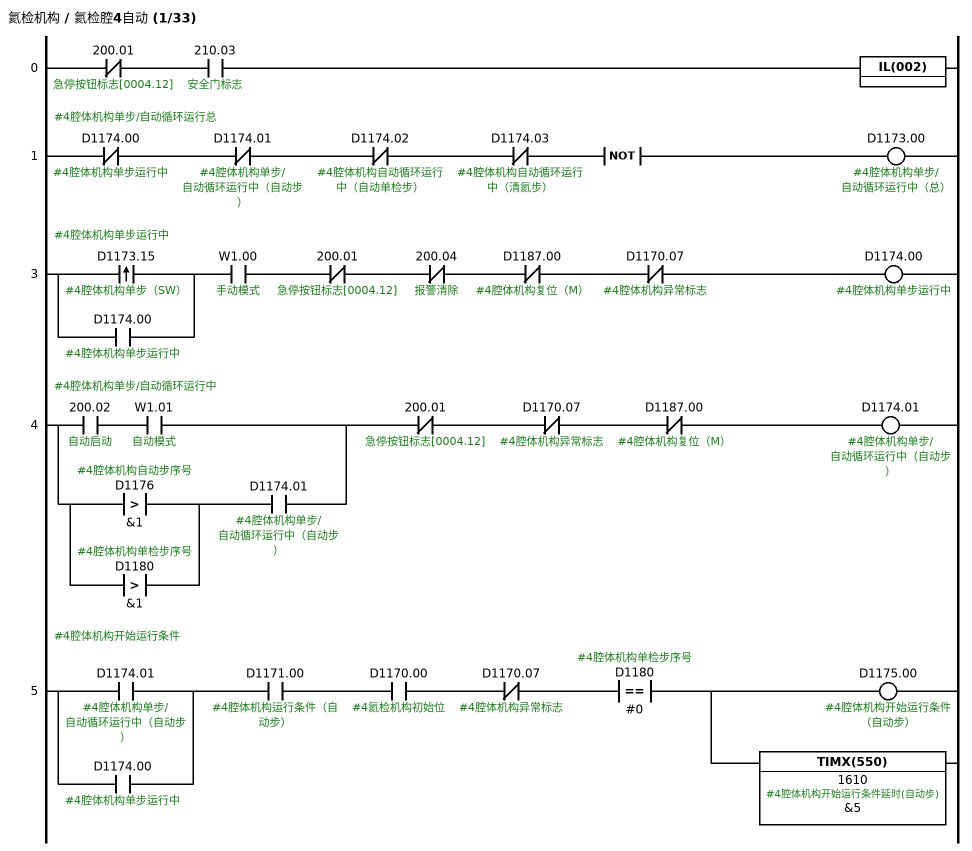
; [picture p336: 氦检机构 / 氦检腔4自动, rungs 0-5]
; rung 0
LDNOT 200.01  ; 急停按钮标志[0004.12]
AND 210.03  ; 安全门标志
IL(002)
; rung 1: #4腔体机构单步/自动循环运行总
LDNOT D1174.00  ; #4腔体机构单步运行中
ANDNOT D1174.01  ; #4腔体机构单步/自动循环运行中（自动步）
ANDNOT D1174.02  ; #4腔体机构自动循环运行中（自动单检步）
ANDNOT D1174.03  ; #4腔体机构自动循环运行中（清氦步）
NOT(520)
OUT D1173.00  ; #4腔体机构单步/自动循环运行中（总）
; rung 2: ******************************* / 自动双检步序 / *******************************
; rung 3: #4腔体机构单步运行中
@LD D1173.15  ; #4腔体机构单步（SW）
OR D1174.00  ; #4腔体机构单步运行中
AND W1.00  ; 手动模式
ANDNOT 200.01  ; 急停按钮标志[0004.12]
ANDNOT 200.04  ; 报警清除
ANDNOT D1187.00  ; #4腔体机构复位（M）
ANDNOT D1170.07  ; #4腔体机构异常标志
OUT D1174.00  ; #4腔体机构单步运行中
; rung 4: #4腔体机构单步/自动循环运行中
LD 200.02  ; 自动启动
AND W1.01  ; 自动模式
LD>L(321) D1176 &1  ; #4腔体机构自动步序号
OR>L(321) D1180 &1  ; #4腔体机构单检步序号
AND D1174.01  ; #4腔体机构单步/自动循环运行中（自动步）
ORLD
ANDNOT 200.01  ; 急停按钮标志[0004.12]
ANDNOT D1170.07  ; #4腔体机构异常标志
ANDNOT D1187.00  ; #4腔体机构复位（M）
OUT D1174.01  ; #4腔体机构单步/自动循环运行中（自动步）
; rung 5: #4腔体机构开始运行条件
LD D1174.01  ; #4腔体机构单步/自动循环运行中（自动步）
OR D1174.00  ; #4腔体机构单步运行中
AND D1171.00  ; #4腔体机构运行条件（自动步）
AND D1170.00  ; #4氦检机构初始位
ANDNOT D1170.07  ; #4腔体机构异常标志
AND=L(301) D1180 #0  ; #4腔体机构单检步序号
OUT D1175.00  ; #4腔体机构开始运行条件（自动步）
TIMX(550) 1610 &5  ; #4腔体机构开始运行条件延时(自动步)

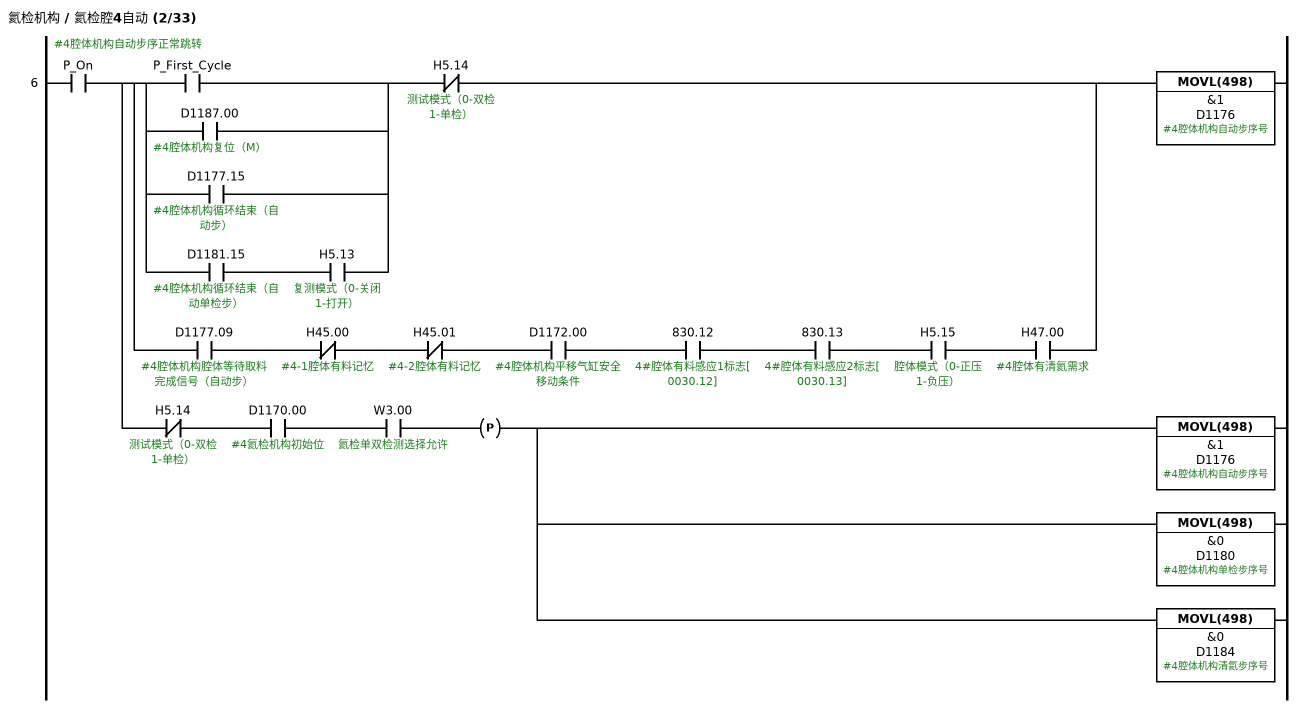
; rung 6: #4腔体机构自动步序正常跳转
LD P_On
OUT TR0
LD P_First_Cycle
OR D1187.00  ; #4腔体机构复位（M）
OR D1177.15  ; #4腔体机构循环结束（自动步）
LD D1181.15  ; #4腔体机构循环结束（自动单检步）
AND H5.13  ; 复测模式（0-关闭 1-打开）
ORLD
ANDNOT H5.14  ; 测试模式（0-双检 1-单检）
LD D1177.09  ; #4腔体机构腔体等待取料完成信号（自动步）  // 负压有清氦需求时，无需回初始位,直接跳回初始步序（D1176.00）
ANDNOT H45.00  ; #4-1腔体有料记忆
ANDNOT H45.01  ; #4-2腔体有料记忆
AND D1172.00  ; #4腔体机构平移气缸安全移动条件
AND 830.12  ; 4#腔体有料感应1标志[0030.12]
AND 830.13  ; 4#腔体有料感应2标志[0030.13]
AND H5.15  ; 腔体模式（0-正压 1-负压）
AND H47.00  ; #4腔体有清氦需求
ORLD
ANDLD
MOVL(498) &1 D1176  ; #4腔体机构自动步序号
LD TR0
ANDNOT H5.14  ; 测试模式（0-双检 1-单检）
AND D1170.00  ; #4氦检机构初始位
AND W3.00  ; 氦检单双检测选择允许
UP(521)
MOVL(498) &1 D1176  ; #4腔体机构自动步序号
MOVL(498) &0 D1180  ; #4腔体机构单检步序号
MOVL(498) &0 D1184  ; #4腔体机构清氦步序号

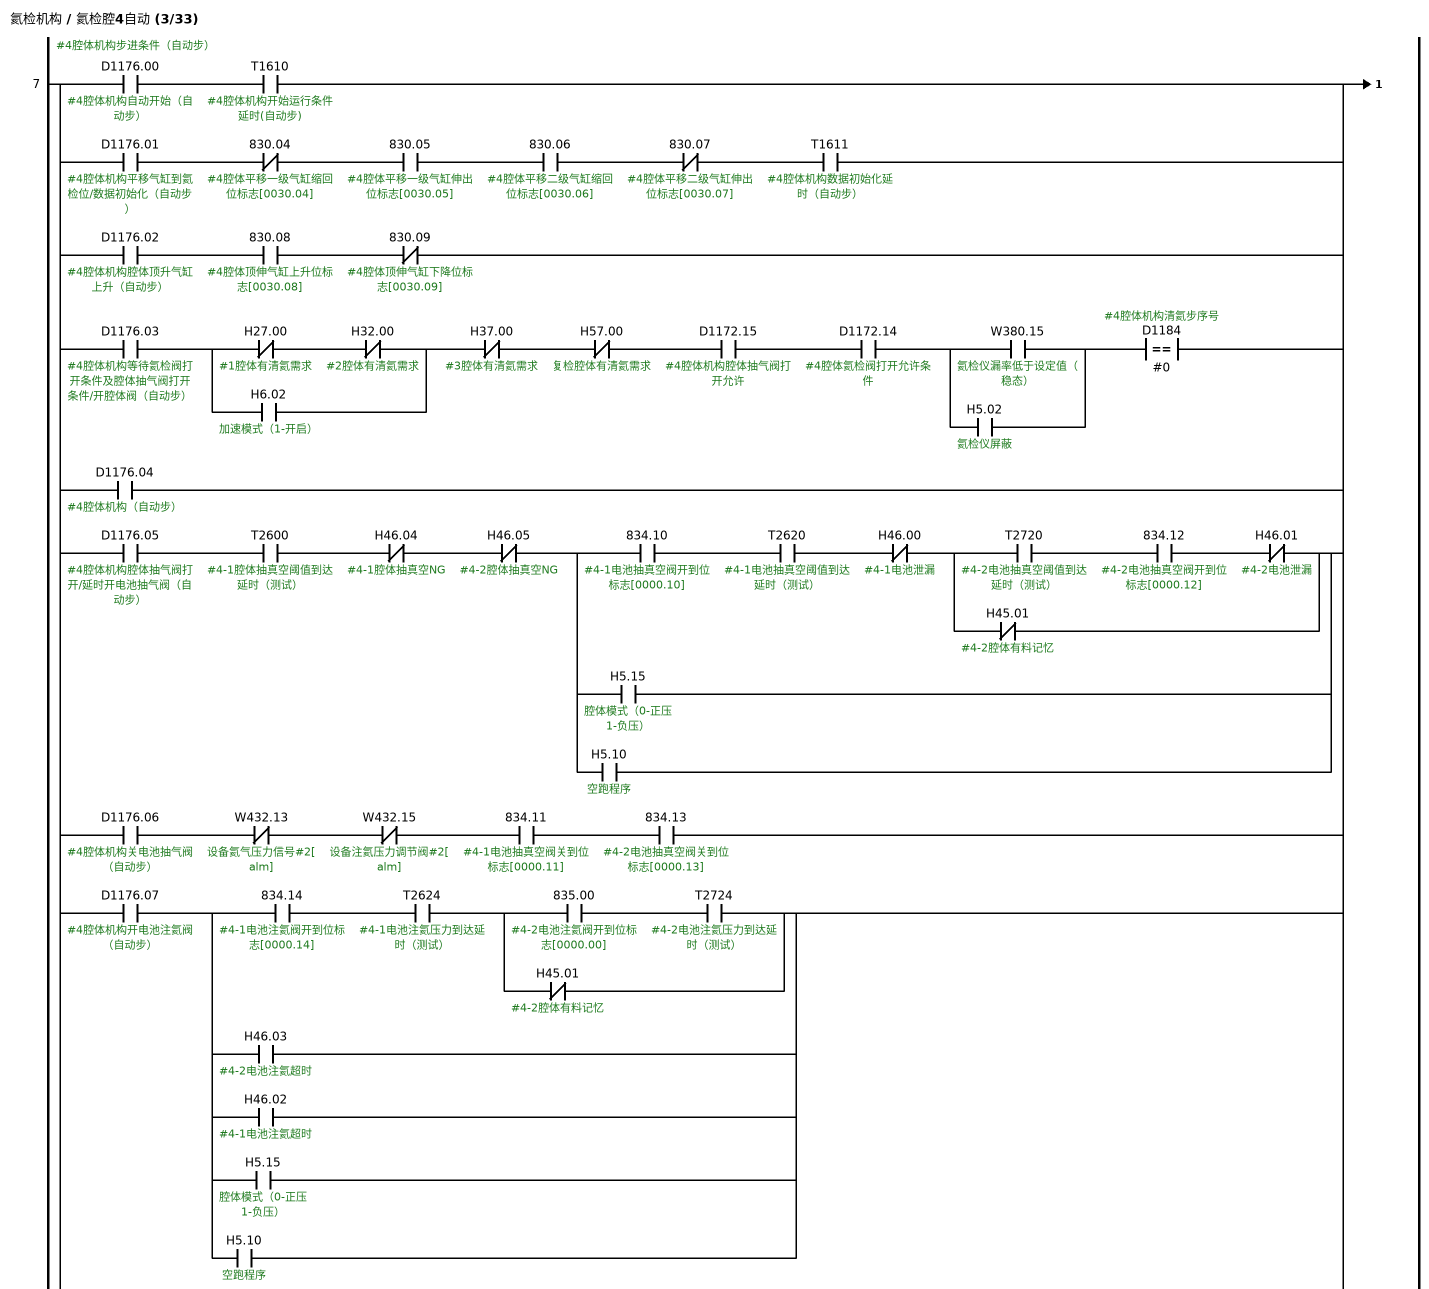

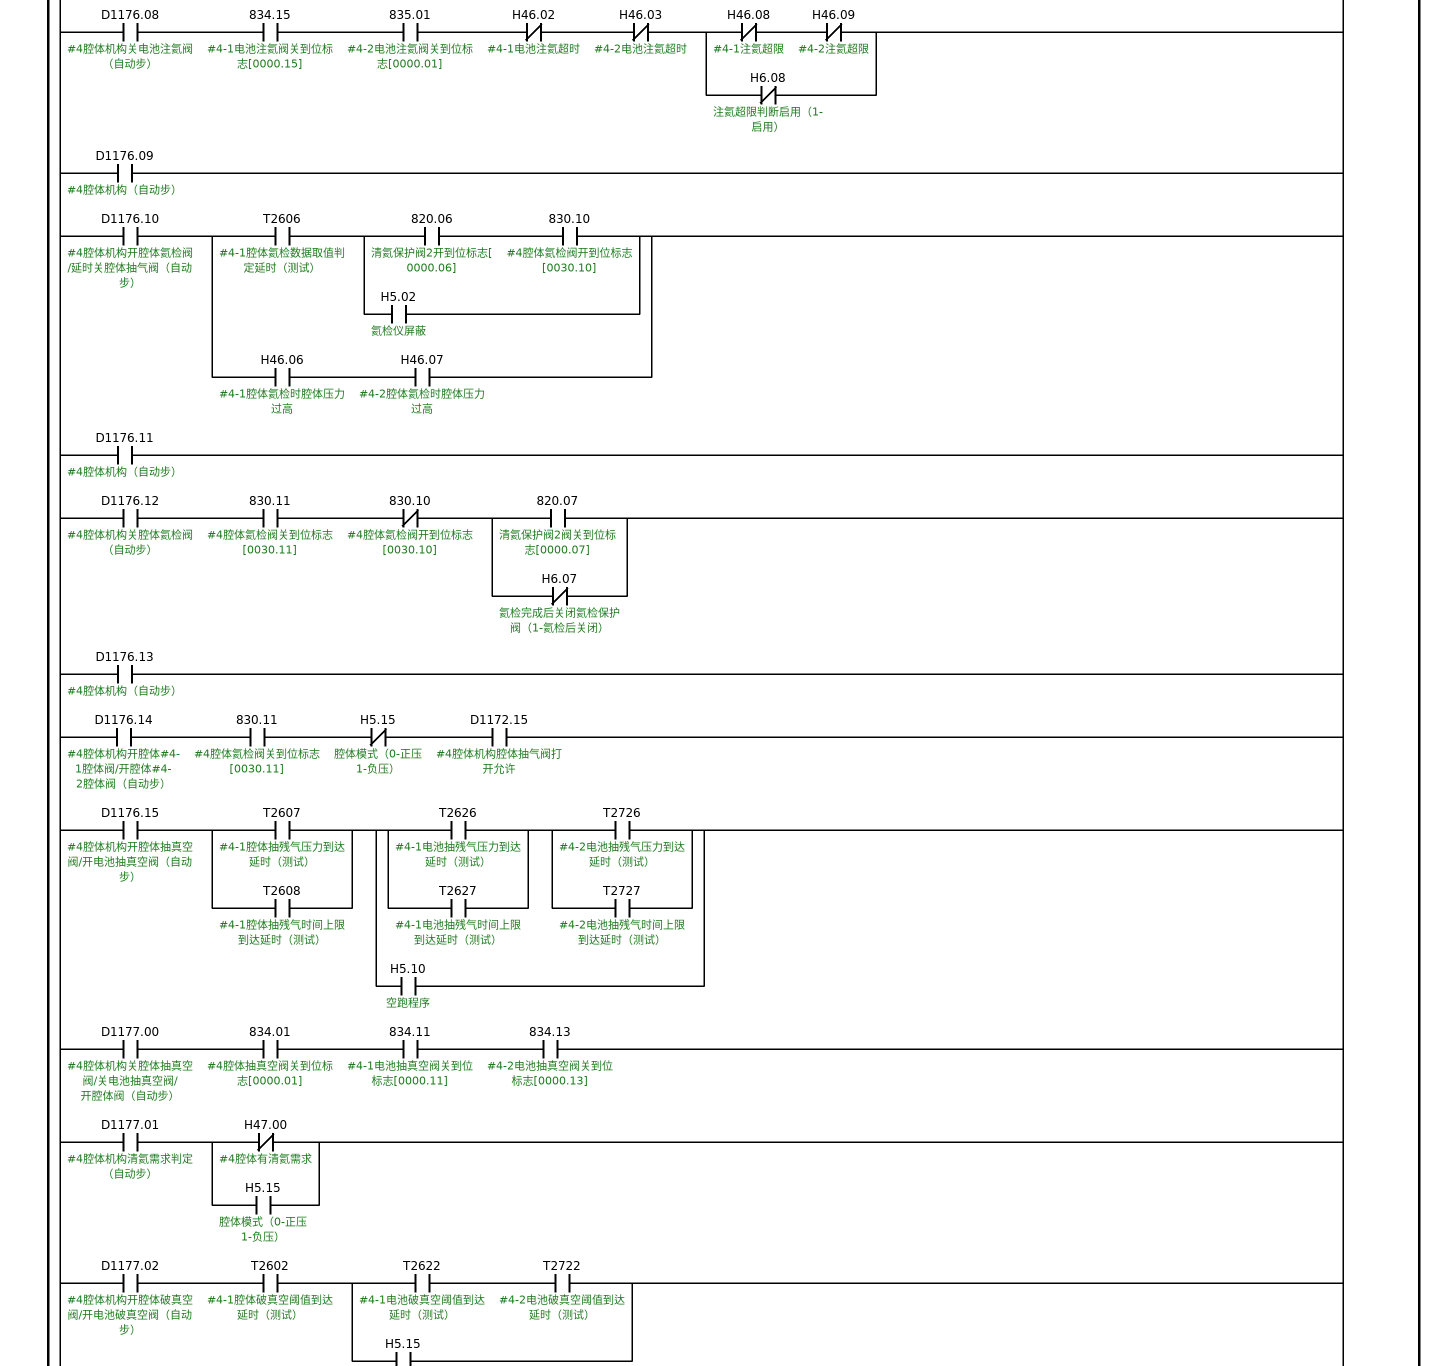

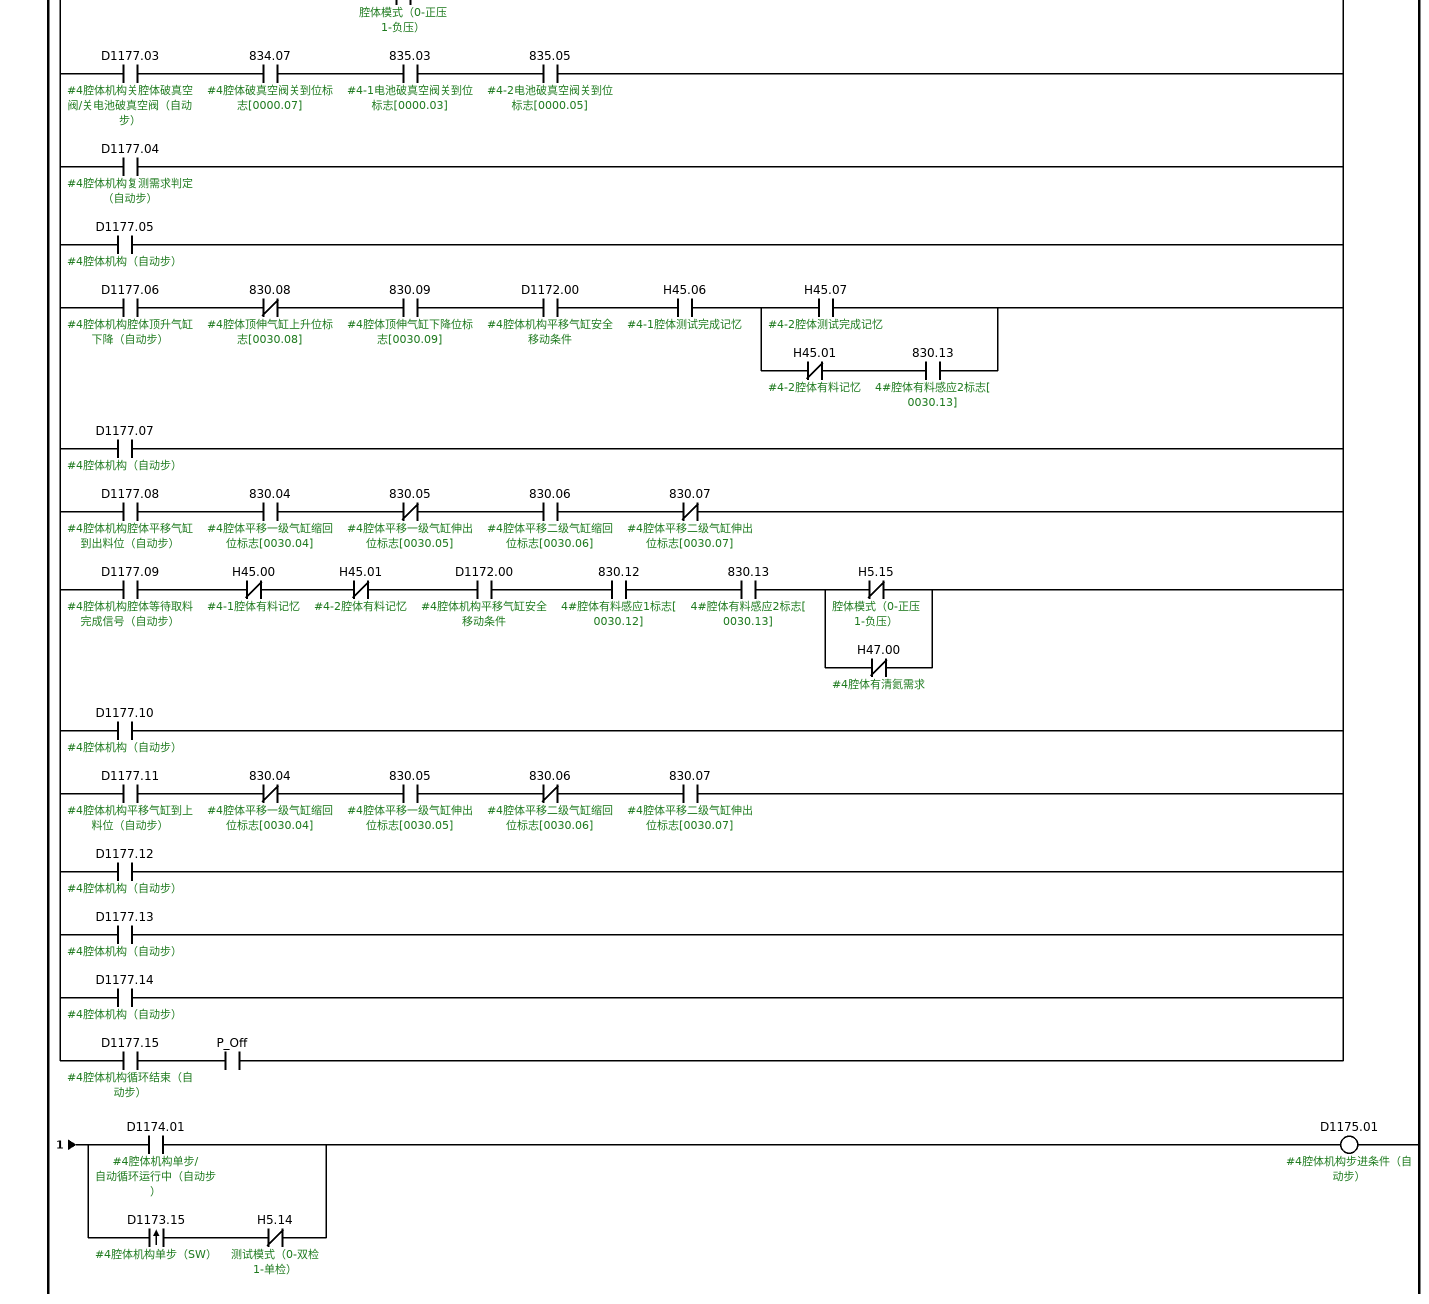
; rung 7: #4腔体机构步进条件（自动步）
LD D1176.00  ; #4腔体机构自动开始（自动步）
AND T1610  ; #4腔体机构开始运行条件延时(自动步)
LD D1176.01  ; #4腔体机构平移气缸到氦检位/数据初始化（自动步）
ANDNOT 830.04  ; #4腔体平移一级气缸缩回位标志[0030.04]
AND 830.05  ; #4腔体平移一级气缸伸出位标志[0030.05]
AND 830.06  ; #4腔体平移二级气缸缩回位标志[0030.06]
ANDNOT 830.07  ; #4腔体平移二级气缸伸出位标志[0030.07]
AND T1611  ; #4腔体机构数据初始化延时（自动步）
ORLD
LD D1176.02  ; #4腔体机构腔体顶升气缸上升（自动步）
AND 830.08  ; #4腔体顶伸气缸上升位标志[0030.08]
ANDNOT 830.09  ; #4腔体顶伸气缸下降位标志[0030.09]
ORLD
LD D1176.03  ; #4腔体机构等待氦检阀打开条件及腔体抽气阀打开条件/开腔体阀（自动步）
LDNOT H27.00  ; #1腔体有清氦需求
ANDNOT H32.00  ; #2腔体有清氦需求
OR H6.02  ; 加速模式（1-开启）
ANDLD
ANDNOT H37.00  ; #3腔体有清氦需求
ANDNOT H57.00  ; 复检腔体有清氦需求
AND D1172.15  ; #4腔体机构腔体抽气阀打开允许
AND D1172.14  ; #4腔体氦检阀打开允许条件
LD W380.15  ; 氦检仪漏率低于设定值（稳态）
OR H5.02  ; 氦检仪屏蔽
ANDLD
AND=L(301) D1184 #0  ; #4腔体机构清氦步序号
ORLD
OR D1176.04  ; #4腔体机构（自动步）
LD D1176.05  ; #4腔体机构腔体抽气阀打开/延时开电池抽气阀（自动步）
AND T2600  ; #4-1腔体抽真空阈值到达延时（测试）
ANDNOT H46.04  ; #4-1腔体抽真空NG
ANDNOT H46.05  ; #4-2腔体抽真空NG
LD 834.10  ; #4-1电池抽真空阀开到位标志[0000.10]
AND T2620  ; #4-1电池抽真空阈值到达延时（测试）
ANDNOT H46.00  ; #4-1电池泄漏
LD T2720  ; #4-2电池抽真空阈值到达延时（测试）
AND 834.12  ; #4-2电池抽真空阀开到位标志[0000.12]
ANDNOT H46.01  ; #4-2电池泄漏
ORNOT H45.01  ; #4-2腔体有料记忆
ANDLD
OR H5.15  ; 腔体模式（0-正压 1-负压）
OR H5.10  ; 空跑程序
ANDLD
ORLD
LD D1176.06  ; #4腔体机构关电池抽气阀（自动步）  // 单个电池出现电池泄漏时，需将对应的腔体阀门关闭
ANDNOT W432.13  ; 设备氦气压力信号#2[alm]
ANDNOT W432.15  ; 设备注氦压力调节阀#2[alm]
AND 834.11  ; #4-1电池抽真空阀关到位标志[0000.11]
AND 834.13  ; #4-2电池抽真空阀关到位标志[0000.13]
ORLD
LD D1176.07  ; #4腔体机构开电池注氦阀（自动步）  // 单个电池出现注氦超时时，需将对应的腔体阀门关闭
LD 834.14  ; #4-1电池注氦阀开到位标志[0000.14]
AND T2624  ; #4-1电池注氦压力到达延时（测试）
LD 835.00  ; #4-2电池注氦阀开到位标志[0000.00]
AND T2724  ; #4-2电池注氦压力到达延时（测试）
ORNOT H45.01  ; #4-2腔体有料记忆
ANDLD
OR H46.03  ; #4-2电池注氦超时
OR H46.02  ; #4-1电池注氦超时
OR H5.15  ; 腔体模式（0-正压 1-负压）
OR H5.10  ; 空跑程序
ANDLD
ORLD
LD D1176.08  ; #4腔体机构关电池注氦阀（自动步）
AND 834.15  ; #4-1电池注氦阀关到位标志[0000.15]
AND 835.01  ; #4-2电池注氦阀关到位标志[0000.01]
ANDNOT H46.02  ; #4-1电池注氦超时
ANDNOT H46.03  ; #4-2电池注氦超时
LDNOT H46.08  ; #4-1注氦超限
ANDNOT H46.09  ; #4-2注氦超限
ORNOT H6.08  ; 注氦超限判断启用（1-启用）
ANDLD
ORLD
OR D1176.09  ; #4腔体机构（自动步）
LD D1176.10  ; #4腔体机构开腔体氦检阀/延时关腔体抽气阀（自动步）
LD T2606  ; #4-1腔体氦检数据取值判定延时（测试）
LD 820.06  ; 清氦保护阀2开到位标志[0000.06]
AND 830.10  ; #4腔体氦检阀开到位标志[0030.10]
OR H5.02  ; 氦检仪屏蔽
ANDLD
LD H46.06  ; #4-1腔体氦检时腔体压力过高
AND H46.07  ; #4-2腔体氦检时腔体压力过高
ORLD
ANDLD
ORLD
OR D1176.11  ; #4腔体机构（自动步）
LD D1176.12  ; #4腔体机构关腔体氦检阀（自动步）
AND 830.11  ; #4腔体氦检阀关到位标志[0030.11]
ANDNOT 830.10  ; #4腔体氦检阀开到位标志[0030.10]
LD 820.07  ; 清氦保护阀2阀关到位标志[0000.07]
ORNOT H6.07  ; 氦检完成后关闭氦检保护阀（1-氦检后关闭）
ANDLD
ORLD
OR D1176.13  ; #4腔体机构（自动步）
LD D1176.14  ; #4腔体机构开腔体#4-1腔体阀/开腔体#4-2腔体阀（自动步）
AND 830.11  ; #4腔体氦检阀关到位标志[0030.11]
ANDNOT H5.15  ; 腔体模式（0-正压 1-负压）
AND D1172.15  ; #4腔体机构腔体抽气阀打开允许
ORLD
LD D1176.15  ; #4腔体机构开腔体抽真空阀/开电池抽真空阀（自动步）
LD T2607  ; #4-1腔体抽残气压力到达延时（测试）
OR T2608  ; #4-1腔体抽残气时间上限到达延时（测试）
ANDLD
LD T2626  ; #4-1电池抽残气压力到达延时（测试）
OR T2627  ; #4-1电池抽残气时间上限到达延时（测试）
LD T2726  ; #4-2电池抽残气压力到达延时（测试）
OR T2727  ; #4-2电池抽残气时间上限到达延时（测试）
ANDLD
OR H5.10  ; 空跑程序
ANDLD
ORLD
LD D1177.00  ; #4腔体机构关腔体抽真空阀/关电池抽真空阀/开腔体阀（自动步）
AND 834.01  ; #4腔体抽真空阀关到位标志[0000.01]
AND 834.11  ; #4-1电池抽真空阀关到位标志[0000.11]
AND 834.13  ; #4-2电池抽真空阀关到位标志[0000.13]
ORLD
LD D1177.01  ; #4腔体机构清氦需求判定（自动步）
LDNOT H47.00  ; #4腔体有清氦需求
OR H5.15  ; 腔体模式（0-正压 1-负压）
ANDLD
ORLD
LD D1177.02  ; #4腔体机构开腔体破真空阀/开电池破真空阀（自动步）
AND T2602  ; #4-1腔体破真空阈值到达延时（测试）
LD T2622  ; #4-1电池破真空阈值到达延时（测试）
AND T2722  ; #4-2电池破真空阈值到达延时（测试）
OR H5.15  ; 腔体模式（0-正压 1-负压）
ANDLD
ORLD
LD D1177.03  ; #4腔体机构关腔体破真空阀/关电池破真空阀（自动步）
AND 834.07  ; #4腔体破真空阀关到位标志[0000.07]
AND 835.03  ; #4-1电池破真空阀关到位标志[0000.03]
AND 835.05  ; #4-2电池破真空阀关到位标志[0000.05]
ORLD
OR D1177.04  ; #4腔体机构复测需求判定（自动步）
OR D1177.05  ; #4腔体机构（自动步）
LD D1177.06  ; #4腔体机构腔体顶升气缸下降（自动步）
ANDNOT 830.08  ; #4腔体顶伸气缸上升位标志[0030.08]
AND 830.09  ; #4腔体顶伸气缸下降位标志[0030.09]
AND D1172.00  ; #4腔体机构平移气缸安全移动条件
AND H45.06  ; #4-1腔体测试完成记忆
LD H45.07  ; #4-2腔体测试完成记忆
LDNOT H45.01  ; #4-2腔体有料记忆
AND 830.13  ; 4#腔体有料感应2标志[0030.13]
ORLD
ANDLD
ORLD
OR D1177.07  ; #4腔体机构（自动步）
LD D1177.08  ; #4腔体机构腔体平移气缸到出料位（自动步）
AND 830.04  ; #4腔体平移一级气缸缩回位标志[0030.04]
ANDNOT 830.05  ; #4腔体平移一级气缸伸出位标志[0030.05]
AND 830.06  ; #4腔体平移二级气缸缩回位标志[0030.06]
ANDNOT 830.07  ; #4腔体平移二级气缸伸出位标志[0030.07]
ORLD
LD D1177.09  ; #4腔体机构腔体等待取料完成信号（自动步）  // 负压有清氦需求时，无需回初始位,直接跳回初始步序（D1176.00）
ANDNOT H45.00  ; #4-1腔体有料记忆
ANDNOT H45.01  ; #4-2腔体有料记忆
AND D1172.00  ; #4腔体机构平移气缸安全移动条件
AND 830.12  ; 4#腔体有料感应1标志[0030.12]
AND 830.13  ; 4#腔体有料感应2标志[0030.13]
LDNOT H5.15  ; 腔体模式（0-正压 1-负压）
ORNOT H47.00  ; #4腔体有清氦需求
ANDLD
ORLD
OR D1177.10  ; #4腔体机构（自动步）
LD D1177.11  ; #4腔体机构平移气缸到上料位（自动步）
ANDNOT 830.04  ; #4腔体平移一级气缸缩回位标志[0030.04]
AND 830.05  ; #4腔体平移一级气缸伸出位标志[0030.05]
ANDNOT 830.06  ; #4腔体平移二级气缸缩回位标志[0030.06]
AND 830.07  ; #4腔体平移二级气缸伸出位标志[0030.07]
ORLD
OR D1177.12  ; #4腔体机构（自动步）
OR D1177.13  ; #4腔体机构（自动步）
OR D1177.14  ; #4腔体机构（自动步）
LD D1177.15  ; #4腔体机构循环结束（自动步）
AND P_Off
ORLD
LD D1174.01  ; #4腔体机构单步/自动循环运行中（自动步）
@LD D1173.15  ; #4腔体机构单步（SW）
ANDNOT H5.14  ; 测试模式（0-双检 1-单检）
ORLD
ANDLD
OUT D1175.01  ; #4腔体机构步进条件（自动步）

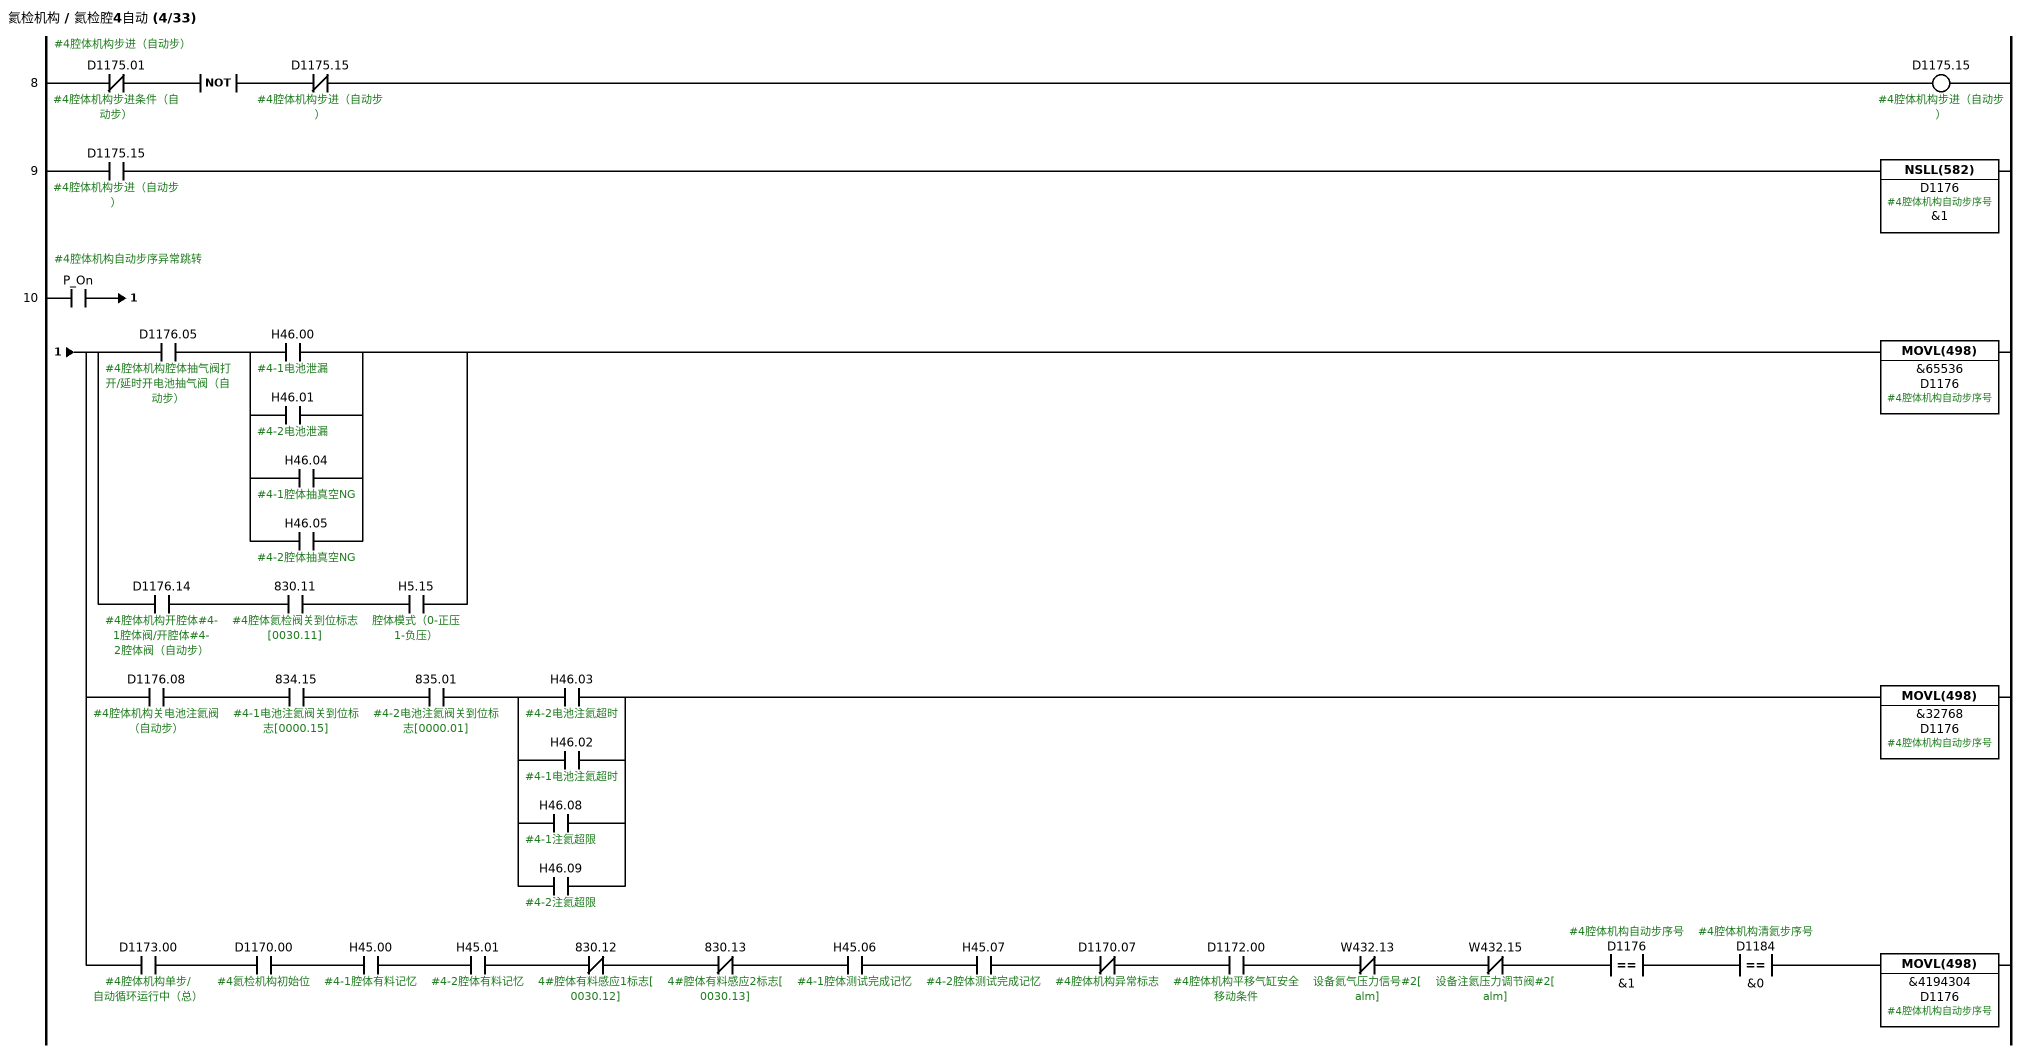
; rung 8: #4腔体机构步进（自动步）
LDNOT D1175.01  ; #4腔体机构步进条件（自动步）
NOT(520)
ANDNOT D1175.15  ; #4腔体机构步进（自动步）
OUT D1175.15  ; #4腔体机构步进（自动步）
; rung 9
LD D1175.15  ; #4腔体机构步进（自动步）
NSLL(582) D1176 &1  ; #4腔体机构自动步序号
; rung 10: #4腔体机构自动步序异常跳转
LD P_On
OUT TR0
LD D1176.05  ; #4腔体机构腔体抽气阀打开/延时开电池抽气阀（自动步）
LD H46.00  ; #4-1电池泄漏
OR H46.01  ; #4-2电池泄漏
OR H46.04  ; #4-1腔体抽真空NG
OR H46.05  ; #4-2腔体抽真空NG
ANDLD
LD D1176.14  ; #4腔体机构开腔体#4-1腔体阀/开腔体#4-2腔体阀（自动步）  // 负压模式不需要进行氦检后抽真空动作
AND 830.11  ; #4腔体氦检阀关到位标志[0030.11]
AND H5.15  ; 腔体模式（0-正压 1-负压）
ORLD
ANDLD
MOVL(498) &65536 D1176  ; #4腔体机构自动步序号  // 出现腔体抽真空NG，双电池抽真空NG，均跳转至自动步序D1067.0
LD TR0
AND D1176.08  ; #4腔体机构关电池注氦阀（自动步）
AND 834.15  ; #4-1电池注氦阀关到位标志[0000.15]
AND 835.01  ; #4-2电池注氦阀关到位标志[0000.01]
LD H46.03  ; #4-2电池注氦超时
OR H46.02  ; #4-1电池注氦超时
OR H46.08  ; #4-1注氦超限
OR H46.09  ; #4-2注氦超限
ANDLD
MOVL(498) &32768 D1176  ; #4腔体机构自动步序号  // 注氦超时需跳转至清氦步序（D1176.15）
LD TR0
AND D1173.00  ; #4腔体机构单步/自动循环运行中（总）
AND D1170.00  ; #4氦检机构初始位
AND H45.00  ; #4-1腔体有料记忆
AND H45.01  ; #4-2腔体有料记忆
ANDNOT 830.12  ; 4#腔体有料感应1标志[0030.12]
ANDNOT 830.13  ; 4#腔体有料感应2标志[0030.13]
AND H45.06  ; #4-1腔体测试完成记忆
AND H45.07  ; #4-2腔体测试完成记忆
ANDNOT D1170.07  ; #4腔体机构异常标志
AND D1172.00  ; #4腔体机构平移气缸安全移动条件
ANDNOT W432.13  ; 设备氦气压力信号#2[alm]
ANDNOT W432.15  ; 设备注氦压力调节阀#2[alm]
AND=L(301) D1176 &1  ; #4腔体机构自动步序号
AND=L(301) D1184 &0  ; #4腔体机构清氦步序号
MOVL(498) &4194304 D1176  ; #4腔体机构自动步序号  // 带料复位时，腔体测试完成后直接跳转至D1177.06
; rung 11: ******************************* / 清氦步序 / *******************************

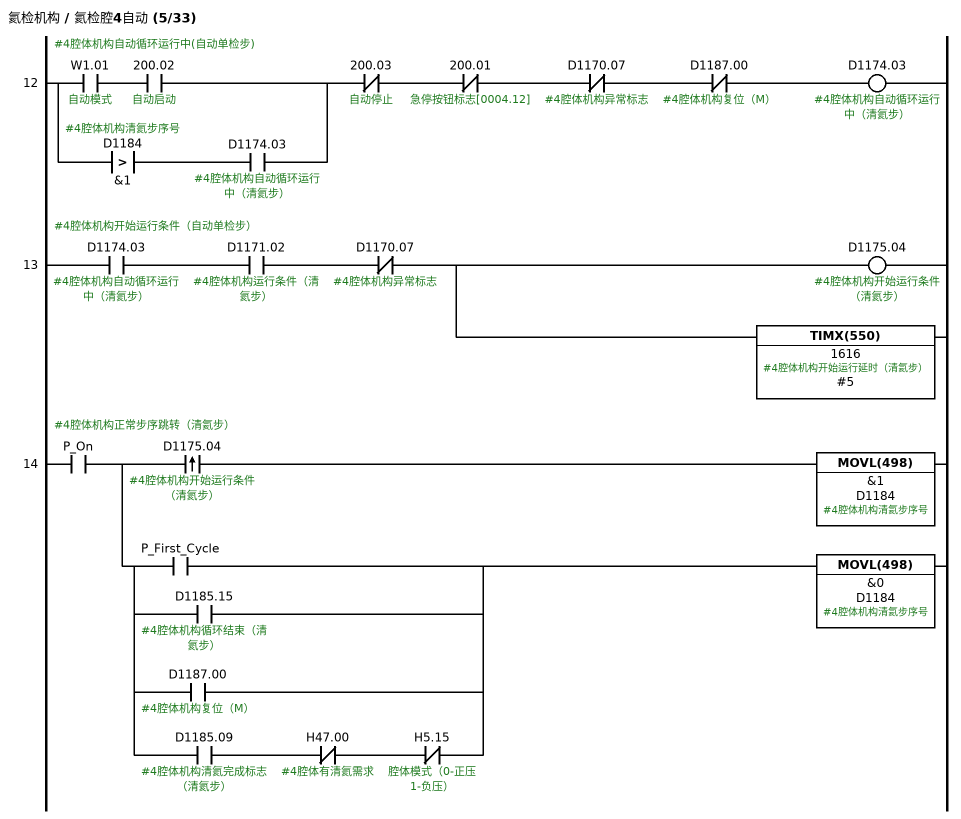
; rung 12: #4腔体机构自动循环运行中(自动单检步)
LD W1.01  ; 自动模式
AND 200.02  ; 自动启动
LD>L(321) D1184 &1  ; #4腔体机构清氦步序号
AND D1174.03  ; #4腔体机构自动循环运行中（清氦步）
ORLD
ANDNOT 200.03  ; 自动停止
ANDNOT 200.01  ; 急停按钮标志[0004.12]
ANDNOT D1170.07  ; #4腔体机构异常标志
ANDNOT D1187.00  ; #4腔体机构复位（M）
OUT D1174.03  ; #4腔体机构自动循环运行中（清氦步）
; rung 13: #4腔体机构开始运行条件（自动单检步）
LD D1174.03  ; #4腔体机构自动循环运行中（清氦步）
AND D1171.02  ; #4腔体机构运行条件（清氦步）
ANDNOT D1170.07  ; #4腔体机构异常标志
OUT D1175.04  ; #4腔体机构开始运行条件（清氦步）
TIMX(550) 1616 #5  ; #4腔体机构开始运行延时（清氦步）
; rung 14: #4腔体机构正常步序跳转（清氦步）
LD P_On
OUT TR0
@AND D1175.04  ; #4腔体机构开始运行条件（清氦步）
MOVL(498) &1 D1184  ; #4腔体机构清氦步序号
LD TR0
LD P_First_Cycle
OR D1185.15  ; #4腔体机构循环结束（清氦步）
OR D1187.00  ; #4腔体机构复位（M）
LD D1185.09  ; #4腔体机构清氦完成标志（清氦步）  // 正压腔体是待料清氦，需跳转回测试步序
ANDNOT H47.00  ; #4腔体有清氦需求
ANDNOT H5.15  ; 腔体模式（0-正压 1-负压）
ORLD
ANDLD
MOVL(498) &0 D1184  ; #4腔体机构清氦步序号

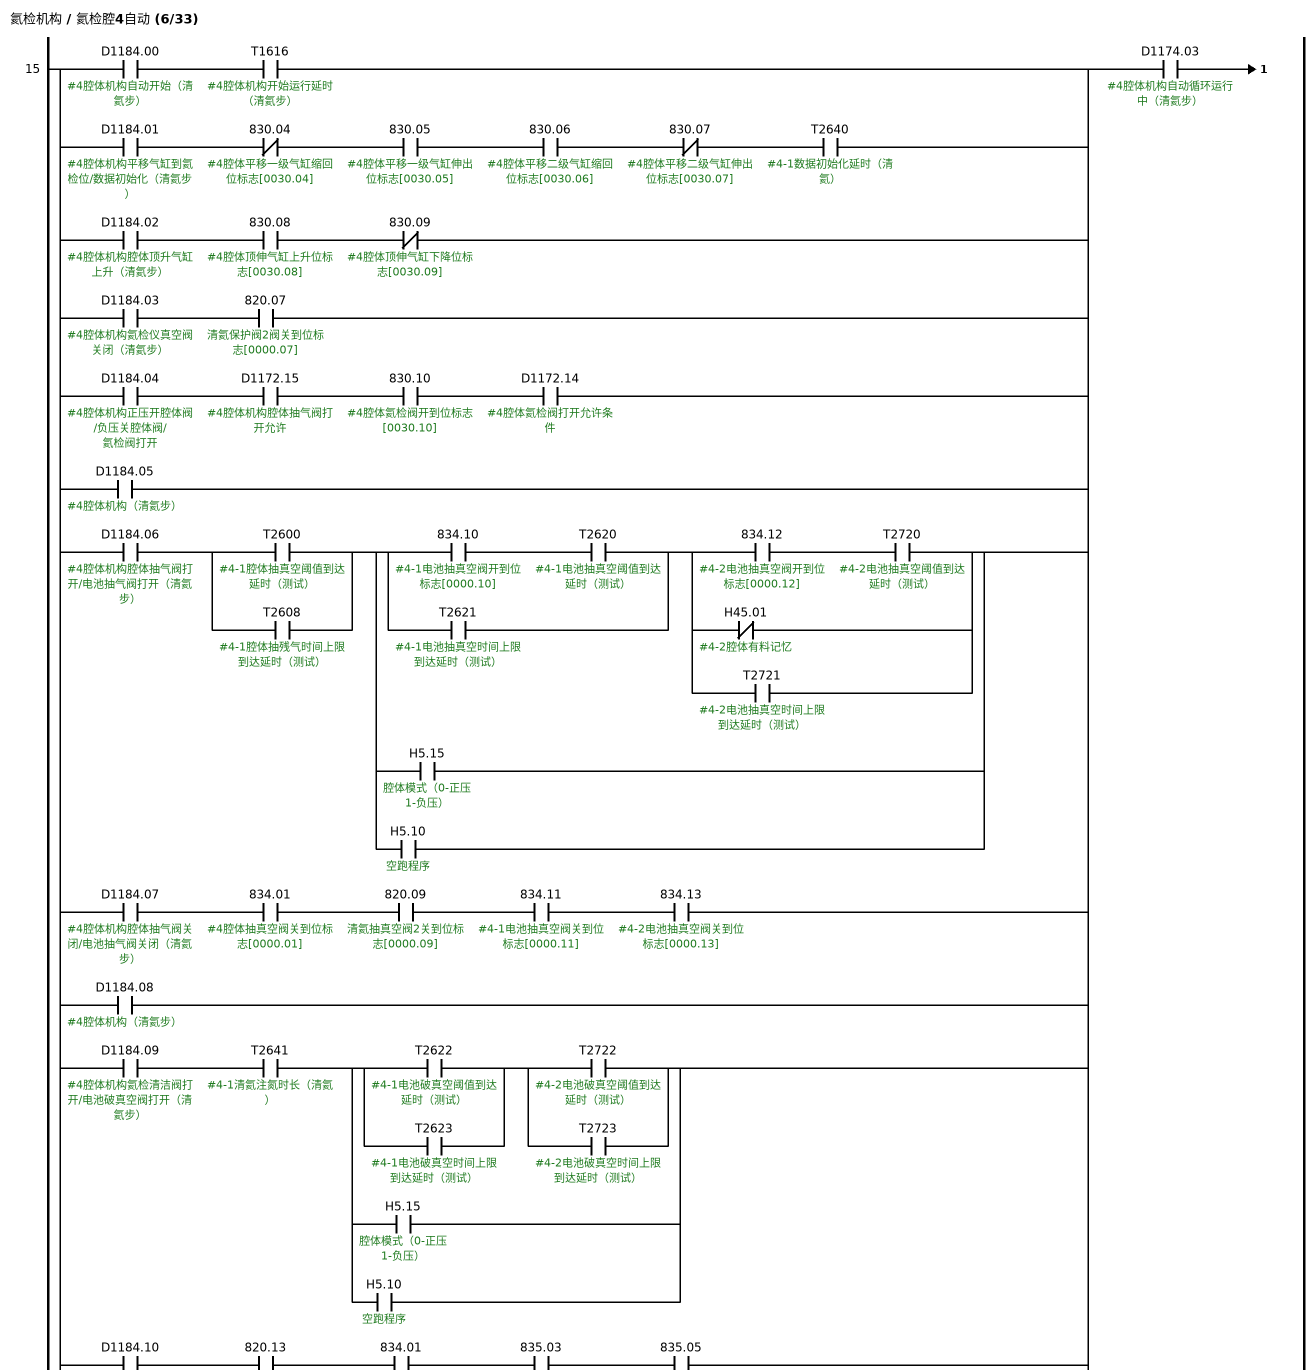

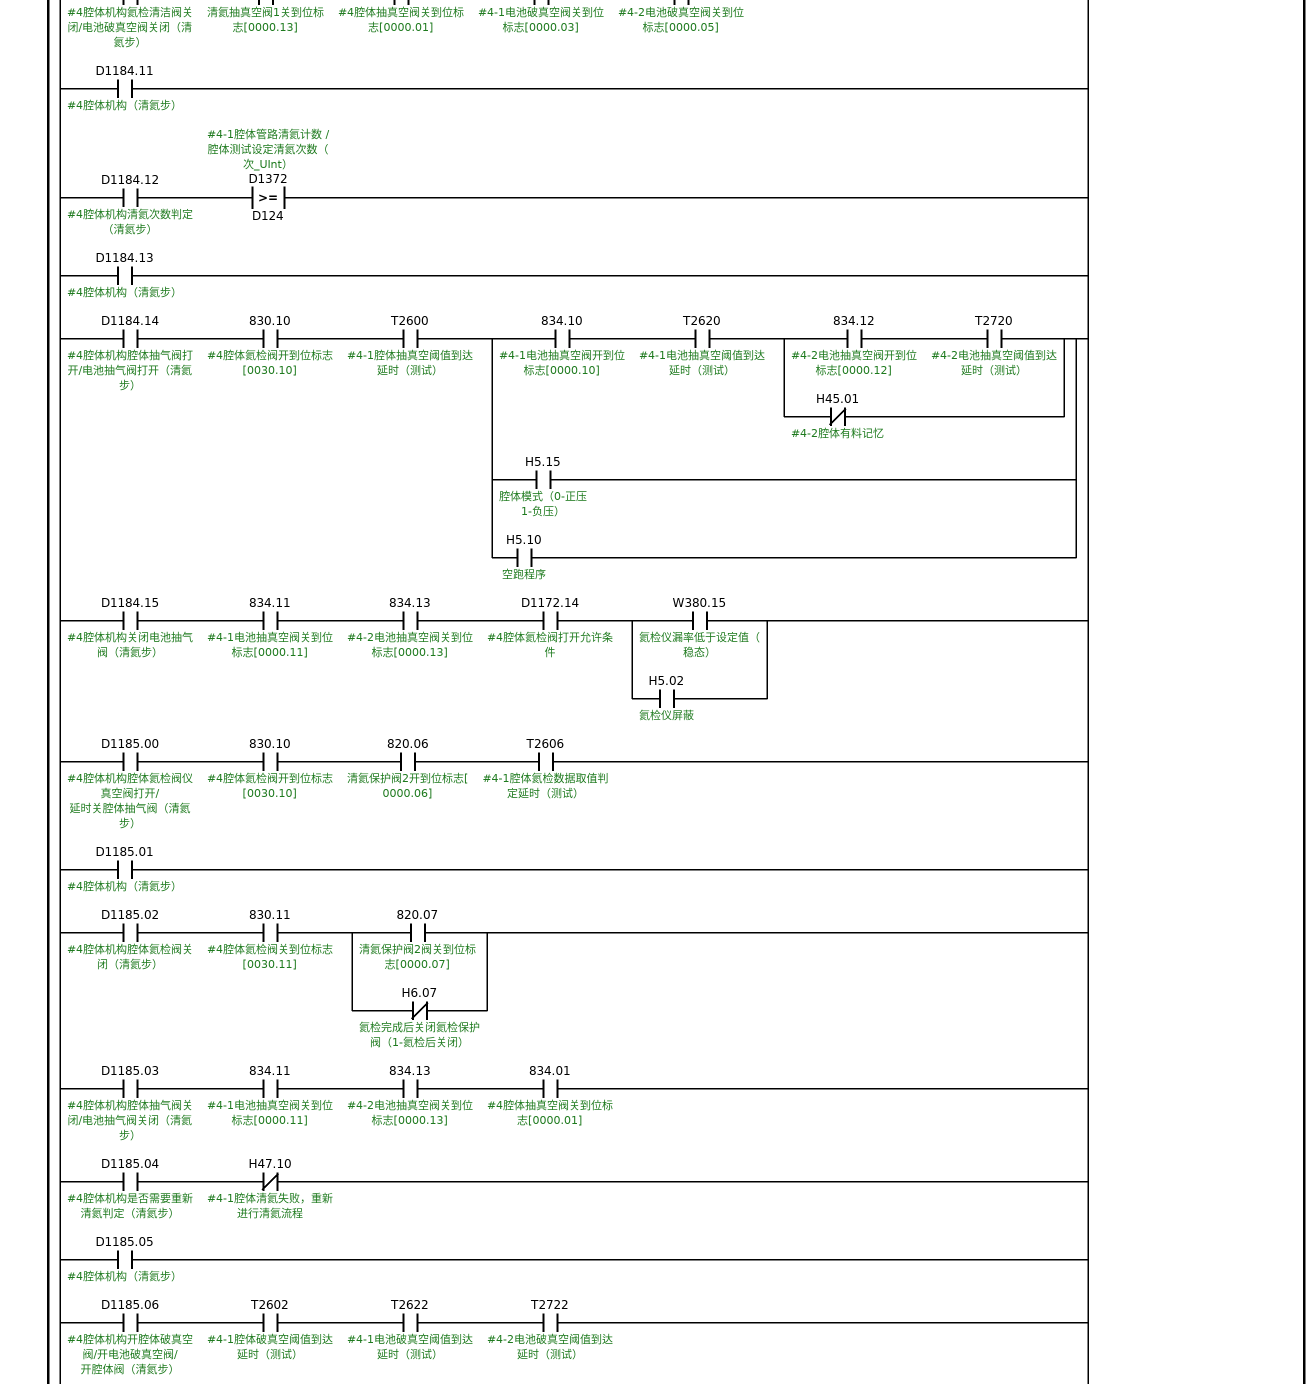

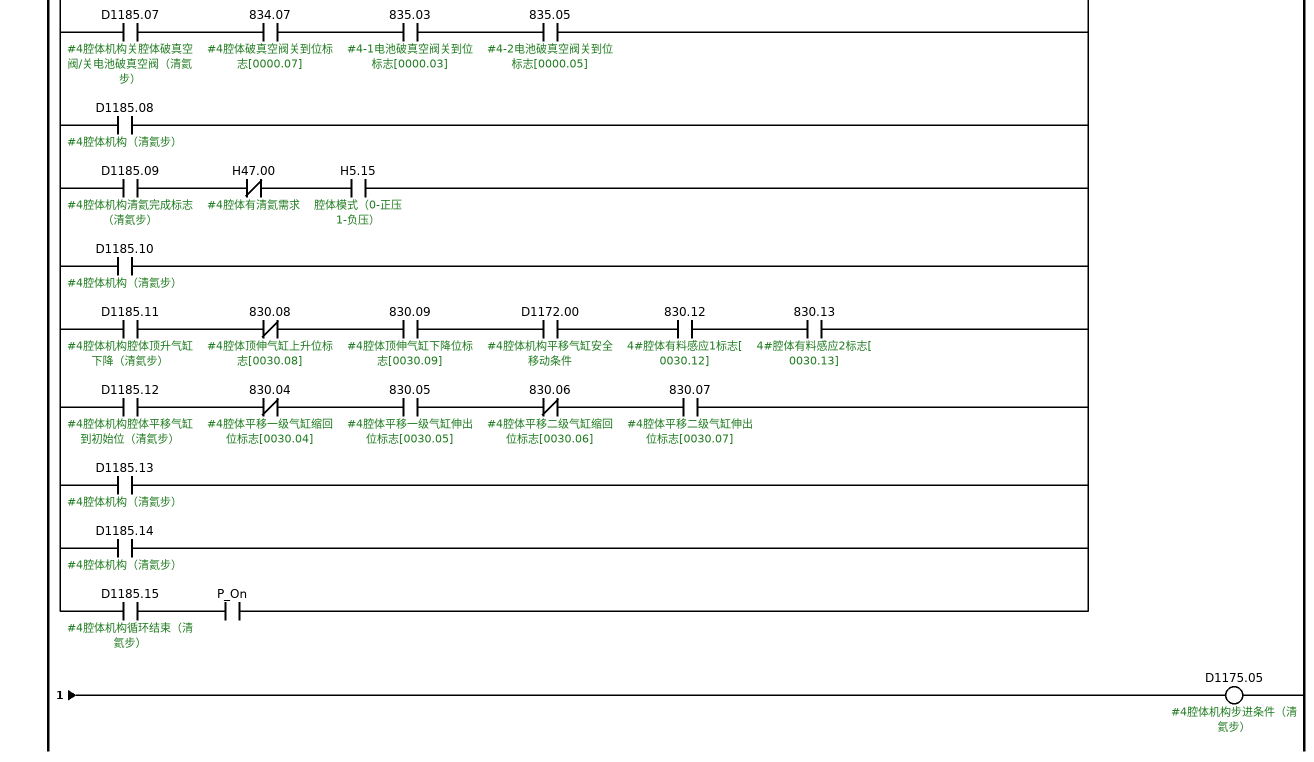
; rung 15
LD D1184.00  ; #4腔体机构自动开始（清氦步）
AND T1616  ; #4腔体机构开始运行延时（清氦步）
LD D1184.01  ; #4腔体机构平移气缸到氦检位/数据初始化（清氦步）
ANDNOT 830.04  ; #4腔体平移一级气缸缩回位标志[0030.04]
AND 830.05  ; #4腔体平移一级气缸伸出位标志[0030.05]
AND 830.06  ; #4腔体平移二级气缸缩回位标志[0030.06]
ANDNOT 830.07  ; #4腔体平移二级气缸伸出位标志[0030.07]
AND T2640  ; #4-1数据初始化延时（清氦）
ORLD
LD D1184.02  ; #4腔体机构腔体顶升气缸上升（清氦步）
AND 830.08  ; #4腔体顶伸气缸上升位标志[0030.08]
ANDNOT 830.09  ; #4腔体顶伸气缸下降位标志[0030.09]
ORLD
LD D1184.03  ; #4腔体机构氦检仪真空阀关闭（清氦步）
AND 820.07  ; 清氦保护阀2阀关到位标志[0000.07]
ORLD
LD D1184.04  ; #4腔体机构正压开腔体阀/负压关腔体阀/氦检阀打开  // 负压模式下，复测前的清氦不允许抽电池
AND D1172.15  ; #4腔体机构腔体抽气阀打开允许
AND 830.10  ; #4腔体氦检阀开到位标志[0030.10]
AND D1172.14  ; #4腔体氦检阀打开允许条件
ORLD
OR D1184.05  ; #4腔体机构（清氦步）
LD D1184.06  ; #4腔体机构腔体抽气阀打开/电池抽气阀打开（清氦步）
LD T2600  ; #4-1腔体抽真空阈值到达延时（测试）
OR T2608  ; #4-1腔体抽残气时间上限到达延时（测试）
ANDLD
LD 834.10  ; #4-1电池抽真空阀开到位标志[0000.10]
AND T2620  ; #4-1电池抽真空阈值到达延时（测试）
OR T2621  ; #4-1电池抽真空时间上限到达延时（测试）
LD 834.12  ; #4-2电池抽真空阀开到位标志[0000.12]
AND T2720  ; #4-2电池抽真空阈值到达延时（测试）
ORNOT H45.01  ; #4-2腔体有料记忆
OR T2721  ; #4-2电池抽真空时间上限到达延时（测试）
ANDLD
OR H5.15  ; 腔体模式（0-正压 1-负压）
OR H5.10  ; 空跑程序
ANDLD
ORLD
LD D1184.07  ; #4腔体机构腔体抽气阀关闭/电池抽气阀关闭（清氦步）
AND 834.01  ; #4腔体抽真空阀关到位标志[0000.01]
AND 820.09  ; 清氦抽真空阀2关到位标志[0000.09]
AND 834.11  ; #4-1电池抽真空阀关到位标志[0000.11]
AND 834.13  ; #4-2电池抽真空阀关到位标志[0000.13]
ORLD
OR D1184.08  ; #4腔体机构（清氦步）
LD D1184.09  ; #4腔体机构氦检清洁阀打开/电池破真空阀打开（清氦步）
AND T2641  ; #4-1清氦注氮时长（清氦）
LD T2622  ; #4-1电池破真空阈值到达延时（测试）
OR T2623  ; #4-1电池破真空时间上限到达延时（测试）
LD T2722  ; #4-2电池破真空阈值到达延时（测试）
OR T2723  ; #4-2电池破真空时间上限到达延时（测试）
ANDLD
OR H5.15  ; 腔体模式（0-正压 1-负压）
OR H5.10  ; 空跑程序
ANDLD
ORLD
LD D1184.10  ; #4腔体机构氦检清洁阀关闭/电池破真空阀关闭（清氦步）
AND 820.13  ; 清氦抽真空阀1关到位标志[0000.13]
AND 834.01  ; #4腔体抽真空阀关到位标志[0000.01]
AND 835.03  ; #4-1电池破真空阀关到位标志[0000.03]
AND 835.05  ; #4-2电池破真空阀关到位标志[0000.05]
ORLD
OR D1184.11  ; #4腔体机构（清氦步）
LD D1184.12  ; #4腔体机构清氦次数判定（清氦步）
AND>=(325) D1372 D124  ; #4-1腔体管路清氦计数, 腔体测试设定清氦次数（次_UInt）
ORLD
OR D1184.13  ; #4腔体机构（清氦步）
LD D1184.14  ; #4腔体机构腔体抽气阀打开/电池抽气阀打开（清氦步）
AND 830.10  ; #4腔体氦检阀开到位标志[0030.10]
AND T2600  ; #4-1腔体抽真空阈值到达延时（测试）
LD 834.10  ; #4-1电池抽真空阀开到位标志[0000.10]
AND T2620  ; #4-1电池抽真空阈值到达延时（测试）
LD 834.12  ; #4-2电池抽真空阀开到位标志[0000.12]
AND T2720  ; #4-2电池抽真空阈值到达延时（测试）
ORNOT H45.01  ; #4-2腔体有料记忆
ANDLD
OR H5.15  ; 腔体模式（0-正压 1-负压）
OR H5.10  ; 空跑程序
ANDLD
ORLD
LD D1184.15  ; #4腔体机构关闭电池抽气阀（清氦步）
AND 834.11  ; #4-1电池抽真空阀关到位标志[0000.11]
AND 834.13  ; #4-2电池抽真空阀关到位标志[0000.13]
AND D1172.14  ; #4腔体氦检阀打开允许条件
LD W380.15  ; 氦检仪漏率低于设定值（稳态）
OR H5.02  ; 氦检仪屏蔽
ANDLD
ORLD
LD D1185.00  ; #4腔体机构腔体氦检阀仪真空阀打开/延时关腔体抽气阀（清氦步）
AND 830.10  ; #4腔体氦检阀开到位标志[0030.10]
AND 820.06  ; 清氦保护阀2开到位标志[0000.06]
AND T2606  ; #4-1腔体氦检数据取值判定延时（测试）
ORLD
OR D1185.01  ; #4腔体机构（清氦步）
LD D1185.02  ; #4腔体机构腔体氦检阀关闭（清氦步）
AND 830.11  ; #4腔体氦检阀关到位标志[0030.11]
LD 820.07  ; 清氦保护阀2阀关到位标志[0000.07]
ORNOT H6.07  ; 氦检完成后关闭氦检保护阀（1-氦检后关闭）
ANDLD
ORLD
LD D1185.03  ; #4腔体机构腔体抽气阀关闭/电池抽气阀关闭（清氦步）
AND 834.11  ; #4-1电池抽真空阀关到位标志[0000.11]
AND 834.13  ; #4-2电池抽真空阀关到位标志[0000.13]
AND 834.01  ; #4腔体抽真空阀关到位标志[0000.01]
ORLD
LD D1185.04  ; #4腔体机构是否需要重新清氦判定（清氦步）
ANDNOT H47.10  ; #4-1腔体清氦失败，重新进行清氦流程  // 清氦失败，重新进行清氦
ORLD
OR D1185.05  ; #4腔体机构（清氦步）
LD D1185.06  ; #4腔体机构开腔体破真空阀/开电池破真空阀/开腔体阀（清氦步）
AND T2602  ; #4-1腔体破真空阈值到达延时（测试）
AND T2622  ; #4-1电池破真空阈值到达延时（测试）
AND T2722  ; #4-2电池破真空阈值到达延时（测试）
ORLD
LD D1185.07  ; #4腔体机构关腔体破真空阀/关电池破真空阀（清氦步）
AND 834.07  ; #4腔体破真空阀关到位标志[0000.07]
AND 835.03  ; #4-1电池破真空阀关到位标志[0000.03]
AND 835.05  ; #4-2电池破真空阀关到位标志[0000.05]
ORLD
OR D1185.08  ; #4腔体机构（清氦步）
LD D1185.09  ; #4腔体机构清氦完成标志（清氦步）  // 正压腔体是待料清氦，需跳转回测试步序
ANDNOT H47.00  ; #4腔体有清氦需求
AND H5.15  ; 腔体模式（0-正压 1-负压）
ORLD
OR D1185.10  ; #4腔体机构（清氦步）
LD D1185.11  ; #4腔体机构腔体顶升气缸下降（清氦步）
ANDNOT 830.08  ; #4腔体顶伸气缸上升位标志[0030.08]
AND 830.09  ; #4腔体顶伸气缸下降位标志[0030.09]
AND D1172.00  ; #4腔体机构平移气缸安全移动条件
AND 830.12  ; 4#腔体有料感应1标志[0030.12]
AND 830.13  ; 4#腔体有料感应2标志[0030.13]
ORLD
LD D1185.12  ; #4腔体机构腔体平移气缸到初始位（清氦步）
ANDNOT 830.04  ; #4腔体平移一级气缸缩回位标志[0030.04]
AND 830.05  ; #4腔体平移一级气缸伸出位标志[0030.05]
ANDNOT 830.06  ; #4腔体平移二级气缸缩回位标志[0030.06]
AND 830.07  ; #4腔体平移二级气缸伸出位标志[0030.07]
ORLD
OR D1185.13  ; #4腔体机构（清氦步）
OR D1185.14  ; #4腔体机构（清氦步）
LD D1185.15  ; #4腔体机构循环结束（清氦步）
AND P_On
ORLD
AND D1174.03  ; #4腔体机构自动循环运行中（清氦步）
OUT D1175.05  ; #4腔体机构步进条件（清氦步）

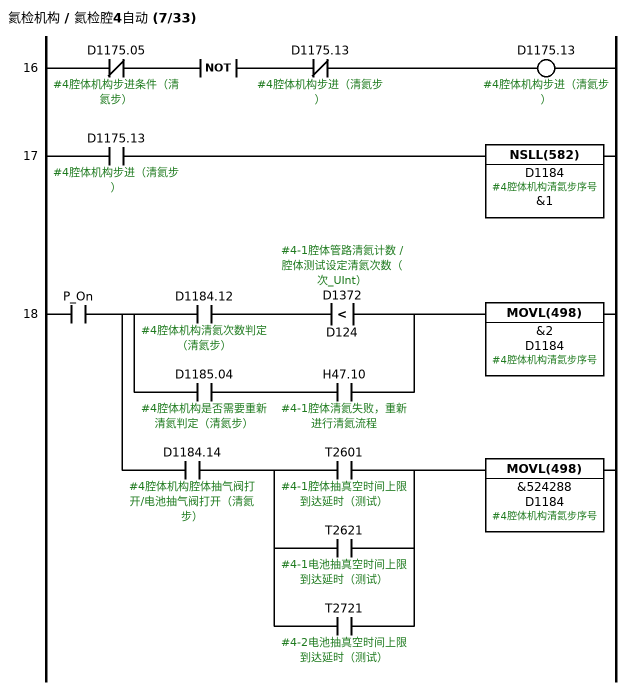
; rung 16
LDNOT D1175.05  ; #4腔体机构步进条件（清氦步）
NOT(520)
ANDNOT D1175.13  ; #4腔体机构步进（清氦步）
OUT D1175.13  ; #4腔体机构步进（清氦步）
; rung 17
LD D1175.13  ; #4腔体机构步进（清氦步）
NSLL(582) D1184 &1  ; #4腔体机构清氦步序号
; rung 18
LD P_On
OUT TR0
LD D1184.12  ; #4腔体机构清氦次数判定（清氦步）
AND<(310) D1372 D124  ; #4-1腔体管路清氦计数, 腔体测试设定清氦次数（次_UInt）
LD D1185.04  ; #4腔体机构是否需要重新清氦判定（清氦步）
AND H47.10  ; #4-1腔体清氦失败，重新进行清氦流程  // 清氦失败，重新进行清氦
ORLD
ANDLD
MOVL(498) &2 D1184  ; #4腔体机构清氦步序号
LD TR0
AND D1184.14  ; #4腔体机构腔体抽气阀打开/电池抽气阀打开（清氦步）
LD T2601  ; #4-1腔体抽真空时间上限到达延时（测试）
OR T2621  ; #4-1电池抽真空时间上限到达延时（测试）
OR T2721  ; #4-2电池抽真空时间上限到达延时（测试）
ANDLD
MOVL(498) &524288 D1184  ; #4腔体机构清氦步序号  // 清氦过程腔体或电池抽气上限达到，均直接判定清氦完成，不进入氦检步序（跳转至D1075.03）

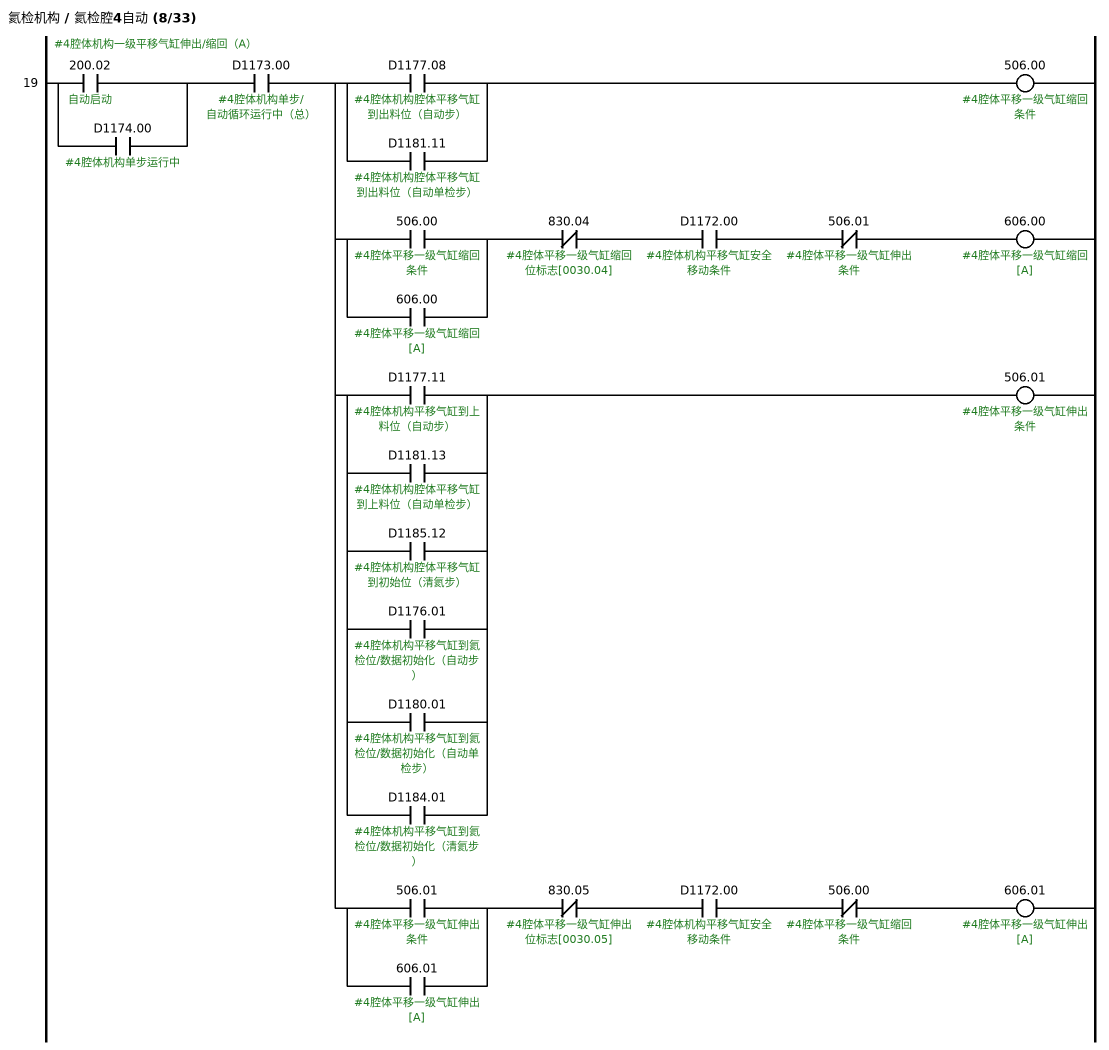
; rung 19: #4腔体机构一级平移气缸伸出/缩回（A）
LD 200.02  ; 自动启动
OR D1174.00  ; #4腔体机构单步运行中
AND D1173.00  ; #4腔体机构单步/自动循环运行中（总）
OUT TR0
LD D1177.08  ; #4腔体机构腔体平移气缸到出料位（自动步）
OR D1181.11  ; #4腔体机构腔体平移气缸到出料位（自动单检步）
ANDLD
OUT 506.00  ; #4腔体平移一级气缸缩回条件
LD TR0
LD 506.00  ; #4腔体平移一级气缸缩回条件
OR 606.00  ; #4腔体平移一级气缸缩回[A]
ANDLD
ANDNOT 830.04  ; #4腔体平移一级气缸缩回位标志[0030.04]
AND D1172.00  ; #4腔体机构平移气缸安全移动条件
ANDNOT 506.01  ; #4腔体平移一级气缸伸出条件
OUT 606.00  ; #4腔体平移一级气缸缩回[A]
LD TR0
LD D1177.11  ; #4腔体机构平移气缸到上料位（自动步）
OR D1181.13  ; #4腔体机构腔体平移气缸到上料位（自动单检步）
OR D1185.12  ; #4腔体机构腔体平移气缸到初始位（清氦步）
OR D1176.01  ; #4腔体机构平移气缸到氦检位/数据初始化（自动步）
OR D1180.01  ; #4腔体机构平移气缸到氦检位/数据初始化（自动单检步）
OR D1184.01  ; #4腔体机构平移气缸到氦检位/数据初始化（清氦步）
ANDLD
OUT 506.01  ; #4腔体平移一级气缸伸出条件
LD TR0
LD 506.01  ; #4腔体平移一级气缸伸出条件
OR 606.01  ; #4腔体平移一级气缸伸出[A]
ANDLD
ANDNOT 830.05  ; #4腔体平移一级气缸伸出位标志[0030.05]
AND D1172.00  ; #4腔体机构平移气缸安全移动条件
ANDNOT 506.00  ; #4腔体平移一级气缸缩回条件
OUT 606.01  ; #4腔体平移一级气缸伸出[A]

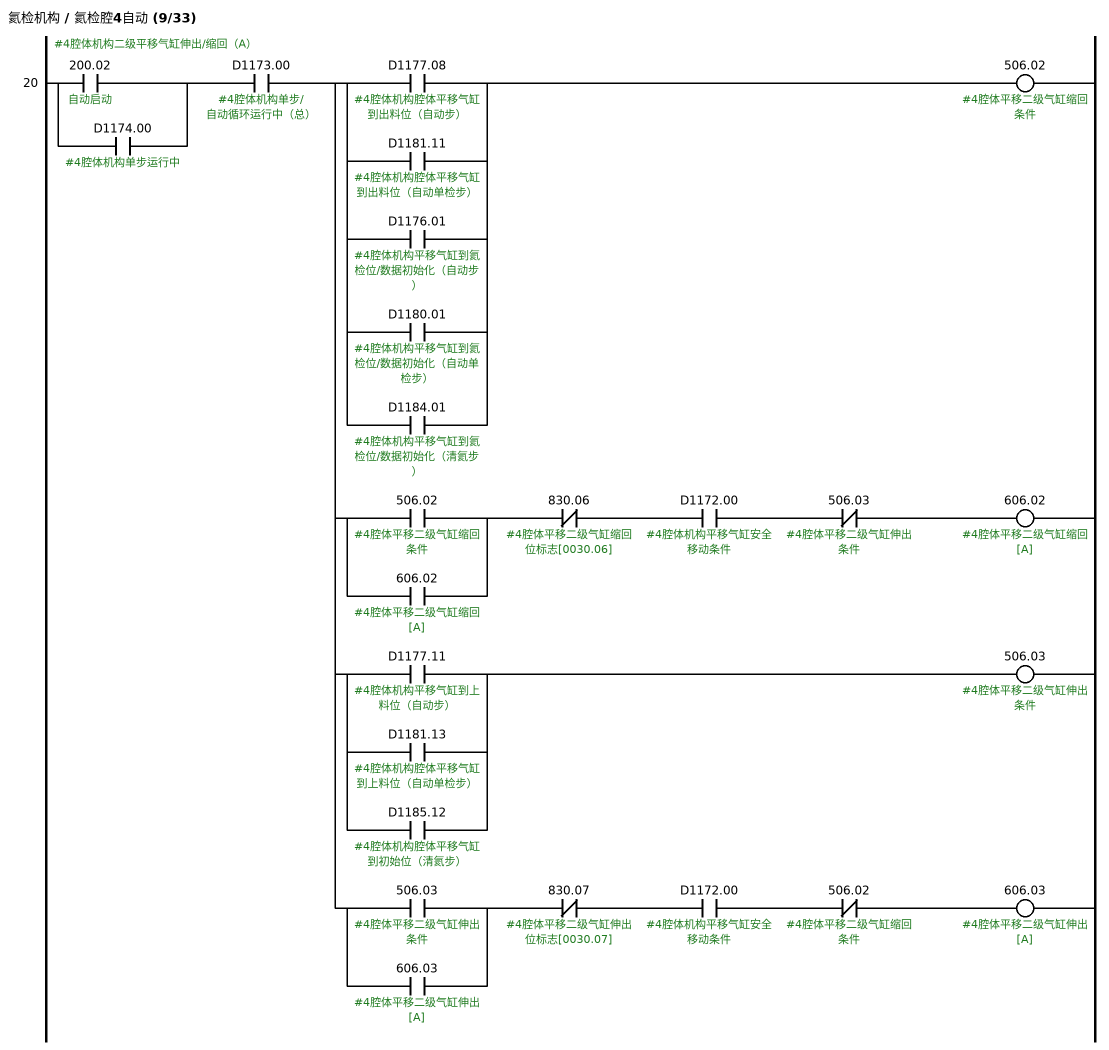
; rung 20: #4腔体机构二级平移气缸伸出/缩回（A）
LD 200.02  ; 自动启动
OR D1174.00  ; #4腔体机构单步运行中
AND D1173.00  ; #4腔体机构单步/自动循环运行中（总）
OUT TR0
LD D1177.08  ; #4腔体机构腔体平移气缸到出料位（自动步）
OR D1181.11  ; #4腔体机构腔体平移气缸到出料位（自动单检步）
OR D1176.01  ; #4腔体机构平移气缸到氦检位/数据初始化（自动步）
OR D1180.01  ; #4腔体机构平移气缸到氦检位/数据初始化（自动单检步）
OR D1184.01  ; #4腔体机构平移气缸到氦检位/数据初始化（清氦步）
ANDLD
OUT 506.02  ; #4腔体平移二级气缸缩回条件
LD TR0
LD 506.02  ; #4腔体平移二级气缸缩回条件
OR 606.02  ; #4腔体平移二级气缸缩回[A]
ANDLD
ANDNOT 830.06  ; #4腔体平移二级气缸缩回位标志[0030.06]
AND D1172.00  ; #4腔体机构平移气缸安全移动条件
ANDNOT 506.03  ; #4腔体平移二级气缸伸出条件
OUT 606.02  ; #4腔体平移二级气缸缩回[A]
LD TR0
LD D1177.11  ; #4腔体机构平移气缸到上料位（自动步）
OR D1181.13  ; #4腔体机构腔体平移气缸到上料位（自动单检步）
OR D1185.12  ; #4腔体机构腔体平移气缸到初始位（清氦步）
ANDLD
OUT 506.03  ; #4腔体平移二级气缸伸出条件
LD TR0
LD 506.03  ; #4腔体平移二级气缸伸出条件
OR 606.03  ; #4腔体平移二级气缸伸出[A]
ANDLD
ANDNOT 830.07  ; #4腔体平移二级气缸伸出位标志[0030.07]
AND D1172.00  ; #4腔体机构平移气缸安全移动条件
ANDNOT 506.02  ; #4腔体平移二级气缸缩回条件
OUT 606.03  ; #4腔体平移二级气缸伸出[A]

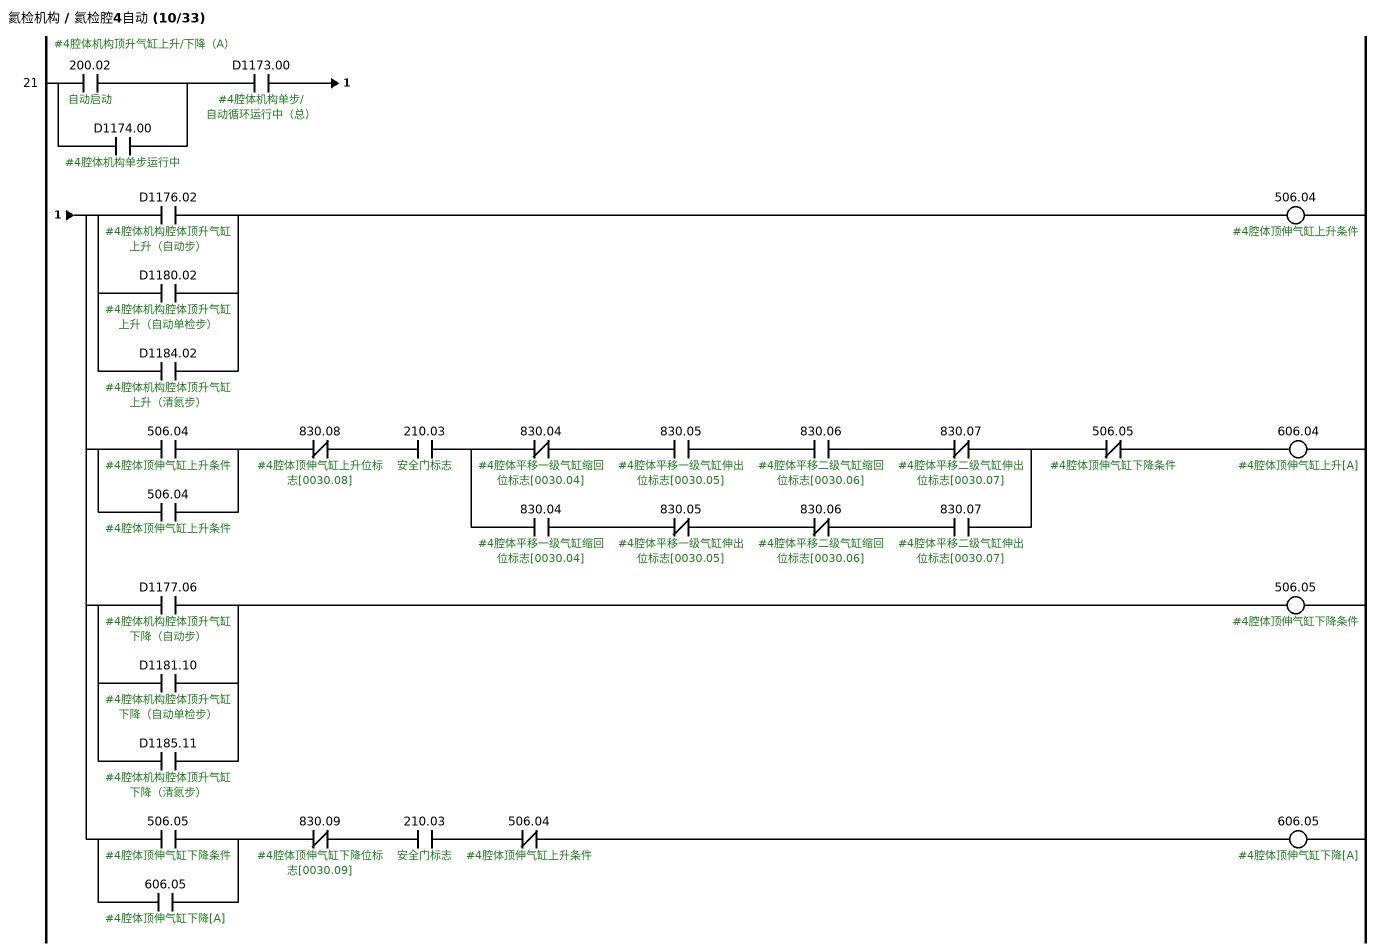
; rung 21: #4腔体机构顶升气缸上升/下降（A）
LD 200.02  ; 自动启动
OR D1174.00  ; #4腔体机构单步运行中
AND D1173.00  ; #4腔体机构单步/自动循环运行中（总）
OUT TR0
LD D1176.02  ; #4腔体机构腔体顶升气缸上升（自动步）
OR D1180.02  ; #4腔体机构腔体顶升气缸上升（自动单检步）
OR D1184.02  ; #4腔体机构腔体顶升气缸上升（清氦步）
ANDLD
OUT 506.04  ; #4腔体顶伸气缸上升条件
LD TR0
LD 506.04  ; #4腔体顶伸气缸上升条件
OR 506.04  ; #4腔体顶伸气缸上升条件
ANDLD
ANDNOT 830.08  ; #4腔体顶伸气缸上升位标志[0030.08]
AND 210.03  ; 安全门标志
LDNOT 830.04  ; #4腔体平移一级气缸缩回位标志[0030.04]
AND 830.05  ; #4腔体平移一级气缸伸出位标志[0030.05]
AND 830.06  ; #4腔体平移二级气缸缩回位标志[0030.06]
ANDNOT 830.07  ; #4腔体平移二级气缸伸出位标志[0030.07]
LD 830.04  ; #4腔体平移一级气缸缩回位标志[0030.04]
ANDNOT 830.05  ; #4腔体平移一级气缸伸出位标志[0030.05]
ANDNOT 830.06  ; #4腔体平移二级气缸缩回位标志[0030.06]
AND 830.07  ; #4腔体平移二级气缸伸出位标志[0030.07]
ORLD
ANDLD
ANDNOT 506.05  ; #4腔体顶伸气缸下降条件
OUT 606.04  ; #4腔体顶伸气缸上升[A]
LD TR0
LD D1177.06  ; #4腔体机构腔体顶升气缸下降（自动步）
OR D1181.10  ; #4腔体机构腔体顶升气缸下降（自动单检步）
OR D1185.11  ; #4腔体机构腔体顶升气缸下降（清氦步）
ANDLD
OUT 506.05  ; #4腔体顶伸气缸下降条件
LD TR0
LD 506.05  ; #4腔体顶伸气缸下降条件
OR 606.05  ; #4腔体顶伸气缸下降[A]
ANDLD
ANDNOT 830.09  ; #4腔体顶伸气缸下降位标志[0030.09]
AND 210.03  ; 安全门标志
ANDNOT 506.04  ; #4腔体顶伸气缸上升条件
OUT 606.05  ; #4腔体顶伸气缸下降[A]

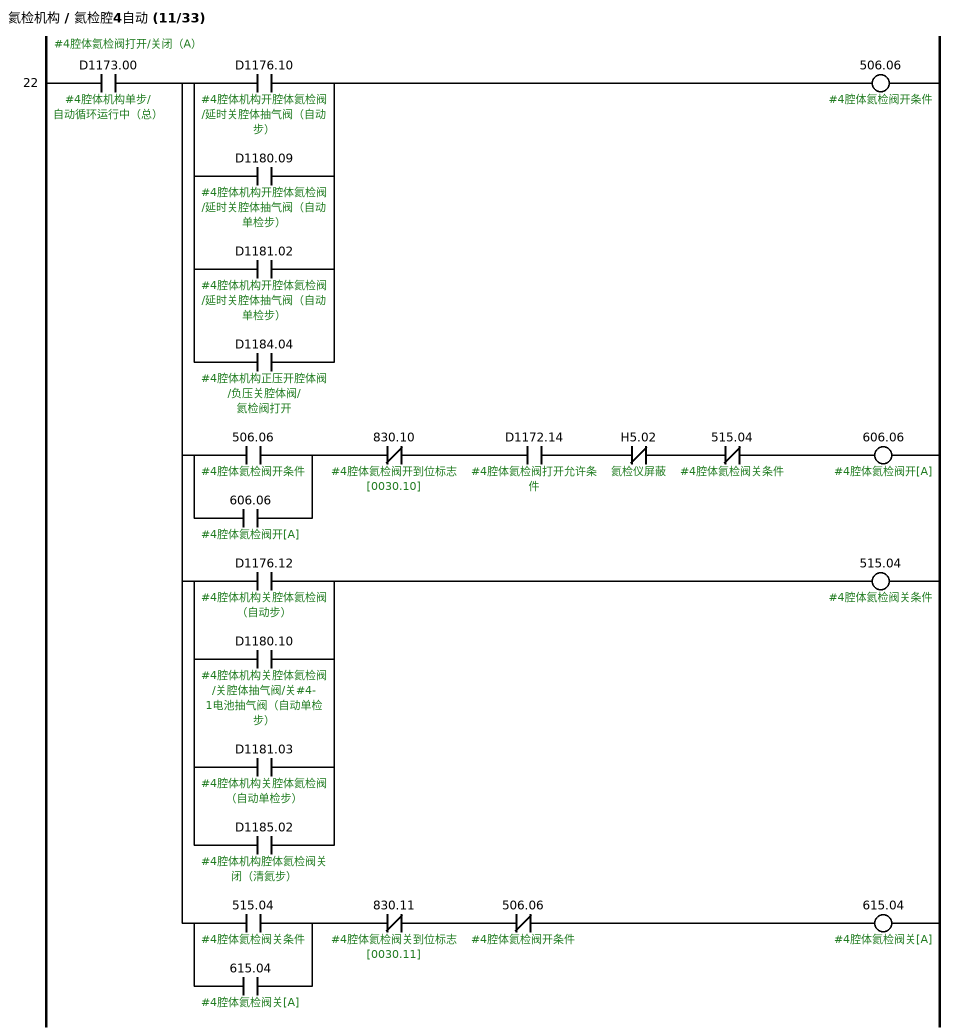
; rung 22: #4腔体氦检阀打开/关闭（A）
LD D1173.00  ; #4腔体机构单步/自动循环运行中（总）
OUT TR0
LD D1176.10  ; #4腔体机构开腔体氦检阀/延时关腔体抽气阀（自动步）
OR D1180.09  ; #4腔体机构开腔体氦检阀/延时关腔体抽气阀（自动单检步）
OR D1181.02  ; #4腔体机构开腔体氦检阀/延时关腔体抽气阀（自动单检步）
OR D1184.04  ; #4腔体机构正压开腔体阀/负压关腔体阀/氦检阀打开
ANDLD
OUT 506.06  ; #4腔体氦检阀开条件
LD TR0
LD 506.06  ; #4腔体氦检阀开条件
OR 606.06  ; #4腔体氦检阀开[A]
ANDLD
ANDNOT 830.10  ; #4腔体氦检阀开到位标志[0030.10]
AND D1172.14  ; #4腔体氦检阀打开允许条件
ANDNOT H5.02  ; 氦检仪屏蔽
ANDNOT 515.04  ; #4腔体氦检阀关条件
OUT 606.06  ; #4腔体氦检阀开[A]
LD TR0
LD D1176.12  ; #4腔体机构关腔体氦检阀（自动步）
OR D1180.10  ; #4腔体机构关腔体氦检阀/关腔体抽气阀/关#4-1电池抽气阀（自动单检步）
OR D1181.03  ; #4腔体机构关腔体氦检阀（自动单检步）
OR D1185.02  ; #4腔体机构腔体氦检阀关闭（清氦步）
ANDLD
OUT 515.04  ; #4腔体氦检阀关条件
LD TR0
LD 515.04  ; #4腔体氦检阀关条件
OR 615.04  ; #4腔体氦检阀关[A]
ANDLD
ANDNOT 830.11  ; #4腔体氦检阀关到位标志[0030.11]
ANDNOT 506.06  ; #4腔体氦检阀开条件
OUT 615.04  ; #4腔体氦检阀关[A]

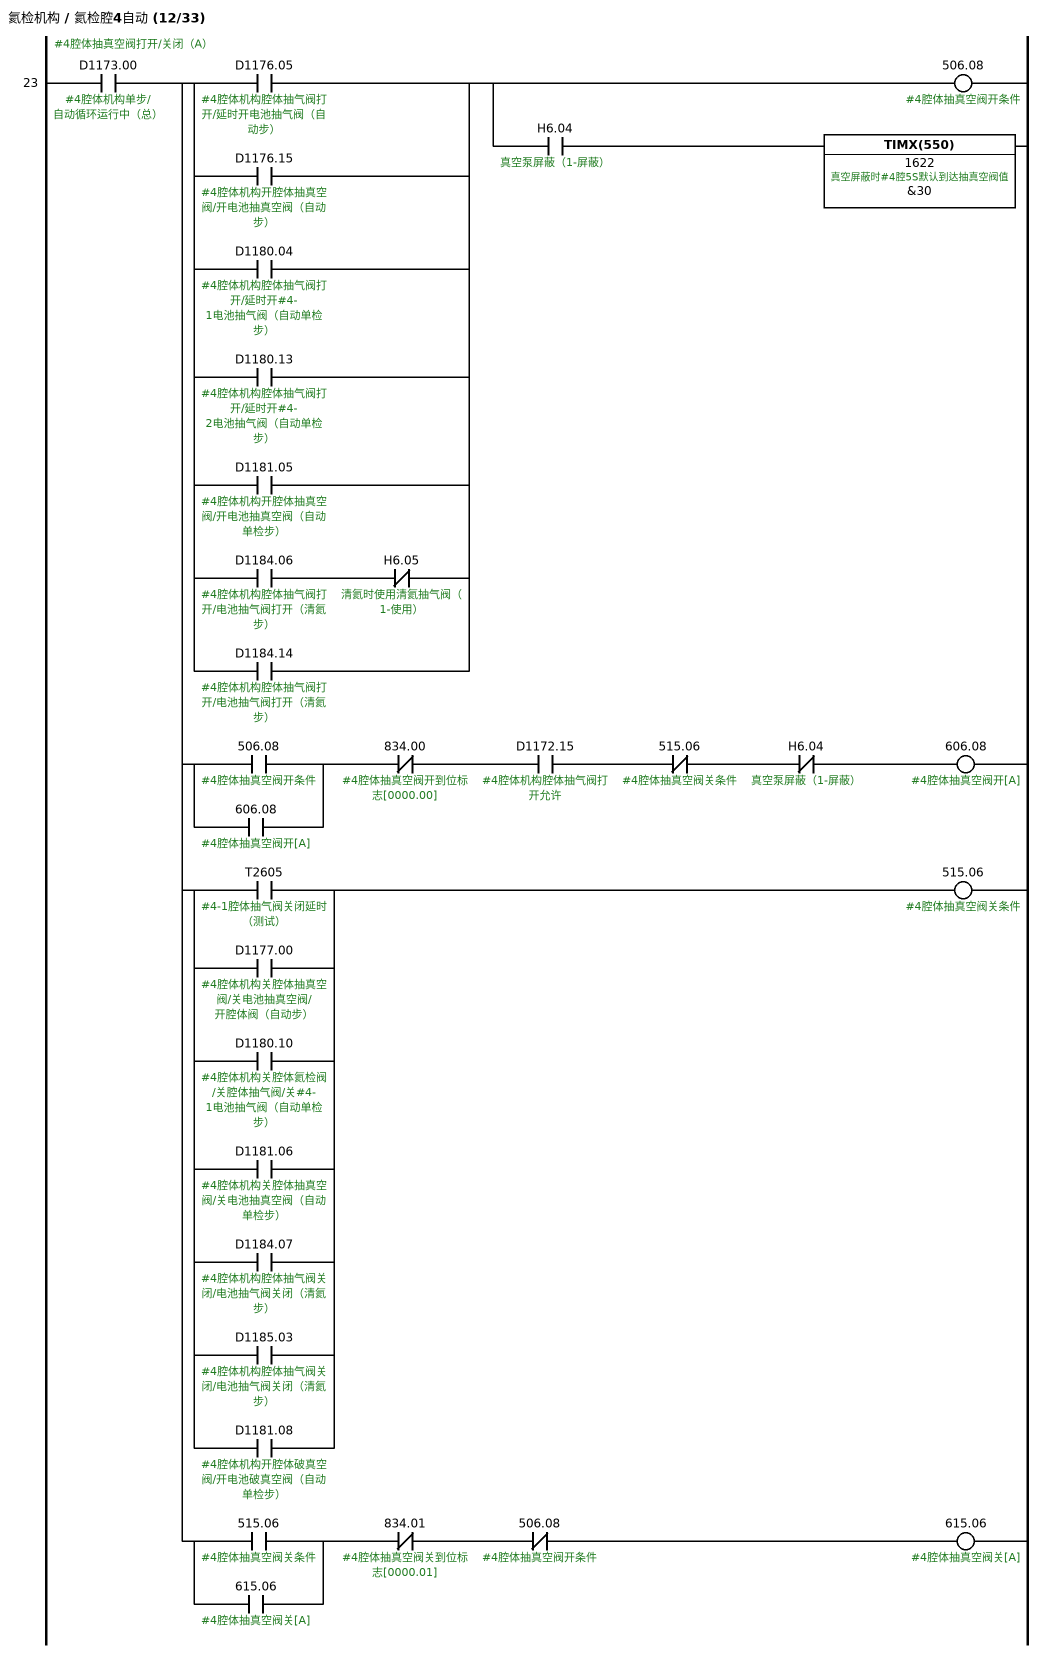
; rung 23: #4腔体抽真空阀打开/关闭（A）
LD D1173.00  ; #4腔体机构单步/自动循环运行中（总）
OUT TR0
LD D1176.05  ; #4腔体机构腔体抽气阀打开/延时开电池抽气阀（自动步）
OR D1176.15  ; #4腔体机构开腔体抽真空阀/开电池抽真空阀（自动步）
OR D1180.04  ; #4腔体机构腔体抽气阀打开/延时开#4-1电池抽气阀（自动单检步）
OR D1180.13  ; #4腔体机构腔体抽气阀打开/延时开#4-2电池抽气阀（自动单检步）
OR D1181.05  ; #4腔体机构开腔体抽真空阀/开电池抽真空阀（自动单检步）
LD D1184.06  ; #4腔体机构腔体抽气阀打开/电池抽气阀打开（清氦步）
ANDNOT H6.05  ; 清氦时使用清氦抽气阀（1-使用）
ORLD
OR D1184.14  ; #4腔体机构腔体抽气阀打开/电池抽气阀打开（清氦步）
ANDLD
OUT 506.08  ; #4腔体抽真空阀开条件
AND H6.04  ; 真空泵屏蔽（1-屏蔽）
TIMX(550) 1622 &30  ; 真空屏蔽时#4腔5S默认到达抽真空阀值
LD TR0
LD 506.08  ; #4腔体抽真空阀开条件
OR 606.08  ; #4腔体抽真空阀开[A]
ANDLD
ANDNOT 834.00  ; #4腔体抽真空阀开到位标志[0000.00]
AND D1172.15  ; #4腔体机构腔体抽气阀打开允许
ANDNOT 515.06  ; #4腔体抽真空阀关条件
ANDNOT H6.04  ; 真空泵屏蔽（1-屏蔽）
OUT 606.08  ; #4腔体抽真空阀开[A]
LD TR0
LD T2605  ; #4-1腔体抽气阀关闭延时（测试）
OR D1177.00  ; #4腔体机构关腔体抽真空阀/关电池抽真空阀/开腔体阀（自动步）
OR D1180.10  ; #4腔体机构关腔体氦检阀/关腔体抽气阀/关#4-1电池抽气阀（自动单检步）
OR D1181.06  ; #4腔体机构关腔体抽真空阀/关电池抽真空阀（自动单检步）
OR D1184.07  ; #4腔体机构腔体抽气阀关闭/电池抽气阀关闭（清氦步）
OR D1185.03  ; #4腔体机构腔体抽气阀关闭/电池抽气阀关闭（清氦步）
OR D1181.08  ; #4腔体机构开腔体破真空阀/开电池破真空阀（自动单检步）
ANDLD
OUT 515.06  ; #4腔体抽真空阀关条件
LD TR0
LD 515.06  ; #4腔体抽真空阀关条件
OR 615.06  ; #4腔体抽真空阀关[A]
ANDLD
ANDNOT 834.01  ; #4腔体抽真空阀关到位标志[0000.01]
ANDNOT 506.08  ; #4腔体抽真空阀开条件
OUT 615.06  ; #4腔体抽真空阀关[A]

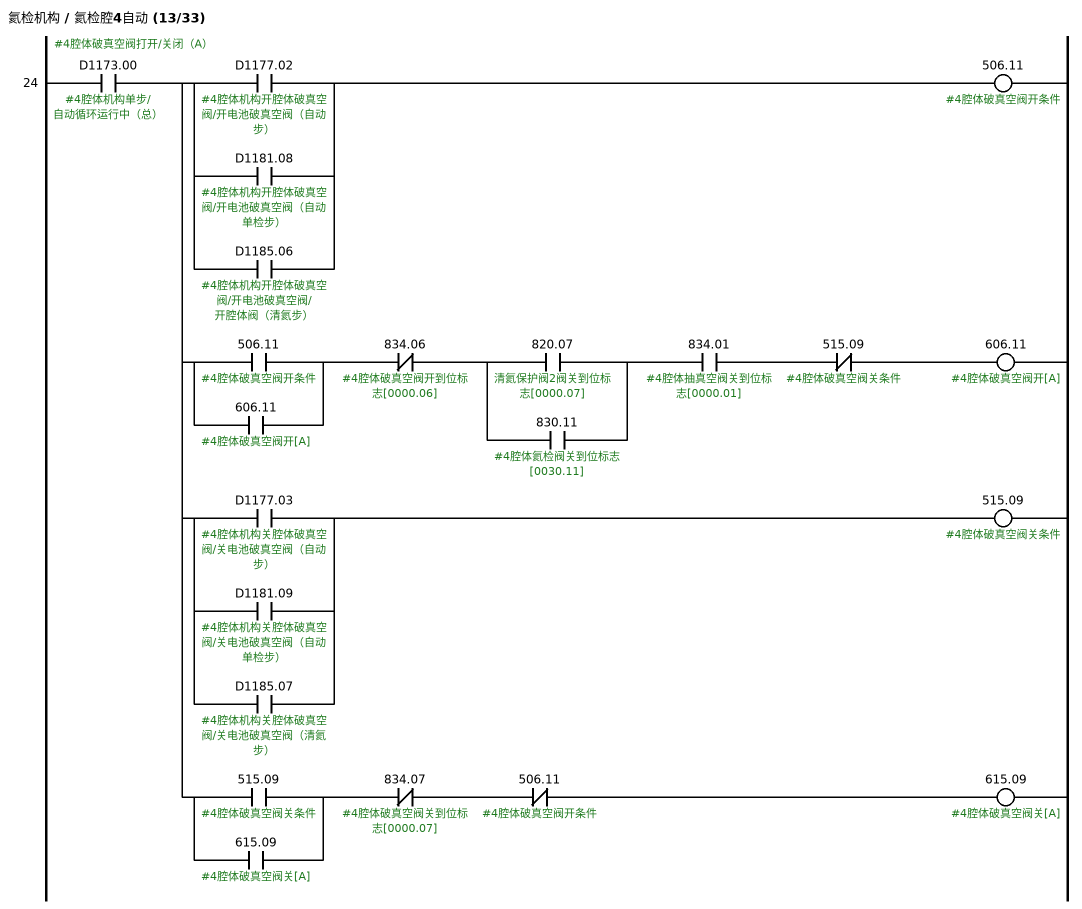
; rung 24: #4腔体破真空阀打开/关闭（A）
LD D1173.00  ; #4腔体机构单步/自动循环运行中（总）
OUT TR0
LD D1177.02  ; #4腔体机构开腔体破真空阀/开电池破真空阀（自动步）
OR D1181.08  ; #4腔体机构开腔体破真空阀/开电池破真空阀（自动单检步）
OR D1185.06  ; #4腔体机构开腔体破真空阀/开电池破真空阀/开腔体阀（清氦步）
ANDLD
OUT 506.11  ; #4腔体破真空阀开条件
LD TR0
LD 506.11  ; #4腔体破真空阀开条件
OR 606.11  ; #4腔体破真空阀开[A]
ANDLD
ANDNOT 834.06  ; #4腔体破真空阀开到位标志[0000.06]
LD 820.07  ; 清氦保护阀2阀关到位标志[0000.07]
OR 830.11  ; #4腔体氦检阀关到位标志[0030.11]
ANDLD
AND 834.01  ; #4腔体抽真空阀关到位标志[0000.01]
ANDNOT 515.09  ; #4腔体破真空阀关条件
OUT 606.11  ; #4腔体破真空阀开[A]
LD TR0
LD D1177.03  ; #4腔体机构关腔体破真空阀/关电池破真空阀（自动步）
OR D1181.09  ; #4腔体机构关腔体破真空阀/关电池破真空阀（自动单检步）
OR D1185.07  ; #4腔体机构关腔体破真空阀/关电池破真空阀（清氦步）
ANDLD
OUT 515.09  ; #4腔体破真空阀关条件
LD TR0
LD 515.09  ; #4腔体破真空阀关条件
OR 615.09  ; #4腔体破真空阀关[A]
ANDLD
ANDNOT 834.07  ; #4腔体破真空阀关到位标志[0000.07]
ANDNOT 506.11  ; #4腔体破真空阀开条件
OUT 615.09  ; #4腔体破真空阀关[A]

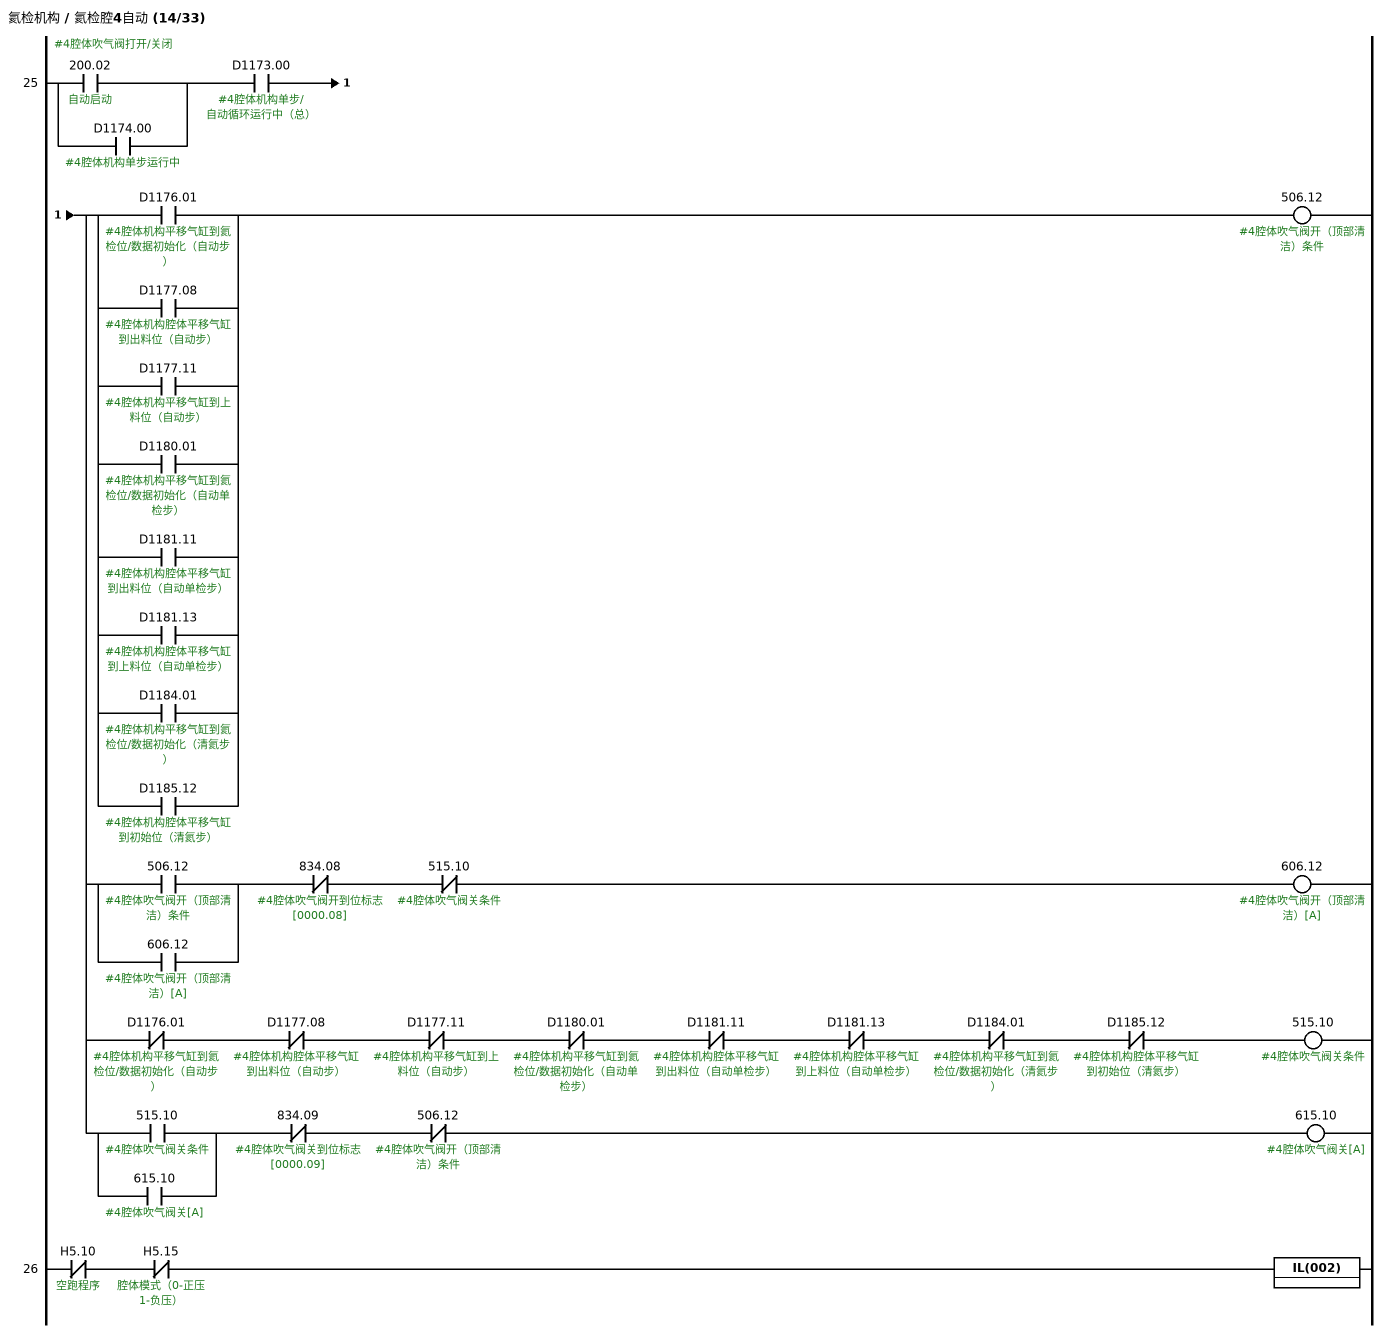
; rung 25: #4腔体吹气阀打开/关闭
LD 200.02  ; 自动启动
OR D1174.00  ; #4腔体机构单步运行中
AND D1173.00  ; #4腔体机构单步/自动循环运行中（总）
OUT TR0
LD D1176.01  ; #4腔体机构平移气缸到氦检位/数据初始化（自动步）
OR D1177.08  ; #4腔体机构腔体平移气缸到出料位（自动步）
OR D1177.11  ; #4腔体机构平移气缸到上料位（自动步）
OR D1180.01  ; #4腔体机构平移气缸到氦检位/数据初始化（自动单检步）
OR D1181.11  ; #4腔体机构腔体平移气缸到出料位（自动单检步）
OR D1181.13  ; #4腔体机构腔体平移气缸到上料位（自动单检步）
OR D1184.01  ; #4腔体机构平移气缸到氦检位/数据初始化（清氦步）
OR D1185.12  ; #4腔体机构腔体平移气缸到初始位（清氦步）
ANDLD
OUT 506.12  ; #4腔体吹气阀开（顶部清洁）条件
LD TR0
LD 506.12  ; #4腔体吹气阀开（顶部清洁）条件
OR 606.12  ; #4腔体吹气阀开（顶部清洁）[A]
ANDLD
ANDNOT 834.08  ; #4腔体吹气阀开到位标志[0000.08]
ANDNOT 515.10  ; #4腔体吹气阀关条件
OUT 606.12  ; #4腔体吹气阀开（顶部清洁）[A]
LD TR0
ANDNOT D1176.01  ; #4腔体机构平移气缸到氦检位/数据初始化（自动步）
ANDNOT D1177.08  ; #4腔体机构腔体平移气缸到出料位（自动步）
ANDNOT D1177.11  ; #4腔体机构平移气缸到上料位（自动步）
ANDNOT D1180.01  ; #4腔体机构平移气缸到氦检位/数据初始化（自动单检步）
ANDNOT D1181.11  ; #4腔体机构腔体平移气缸到出料位（自动单检步）
ANDNOT D1181.13  ; #4腔体机构腔体平移气缸到上料位（自动单检步）
ANDNOT D1184.01  ; #4腔体机构平移气缸到氦检位/数据初始化（清氦步）
ANDNOT D1185.12  ; #4腔体机构腔体平移气缸到初始位（清氦步）
OUT 515.10  ; #4腔体吹气阀关条件
LD TR0
LD 515.10  ; #4腔体吹气阀关条件
OR 615.10  ; #4腔体吹气阀关[A]
ANDLD
ANDNOT 834.09  ; #4腔体吹气阀关到位标志[0000.09]
ANDNOT 506.12  ; #4腔体吹气阀开（顶部清洁）条件
OUT 615.10  ; #4腔体吹气阀关[A]
; rung 26
LDNOT H5.10  ; 空跑程序
ANDNOT H5.15  ; 腔体模式（0-正压 1-负压）
IL(002)

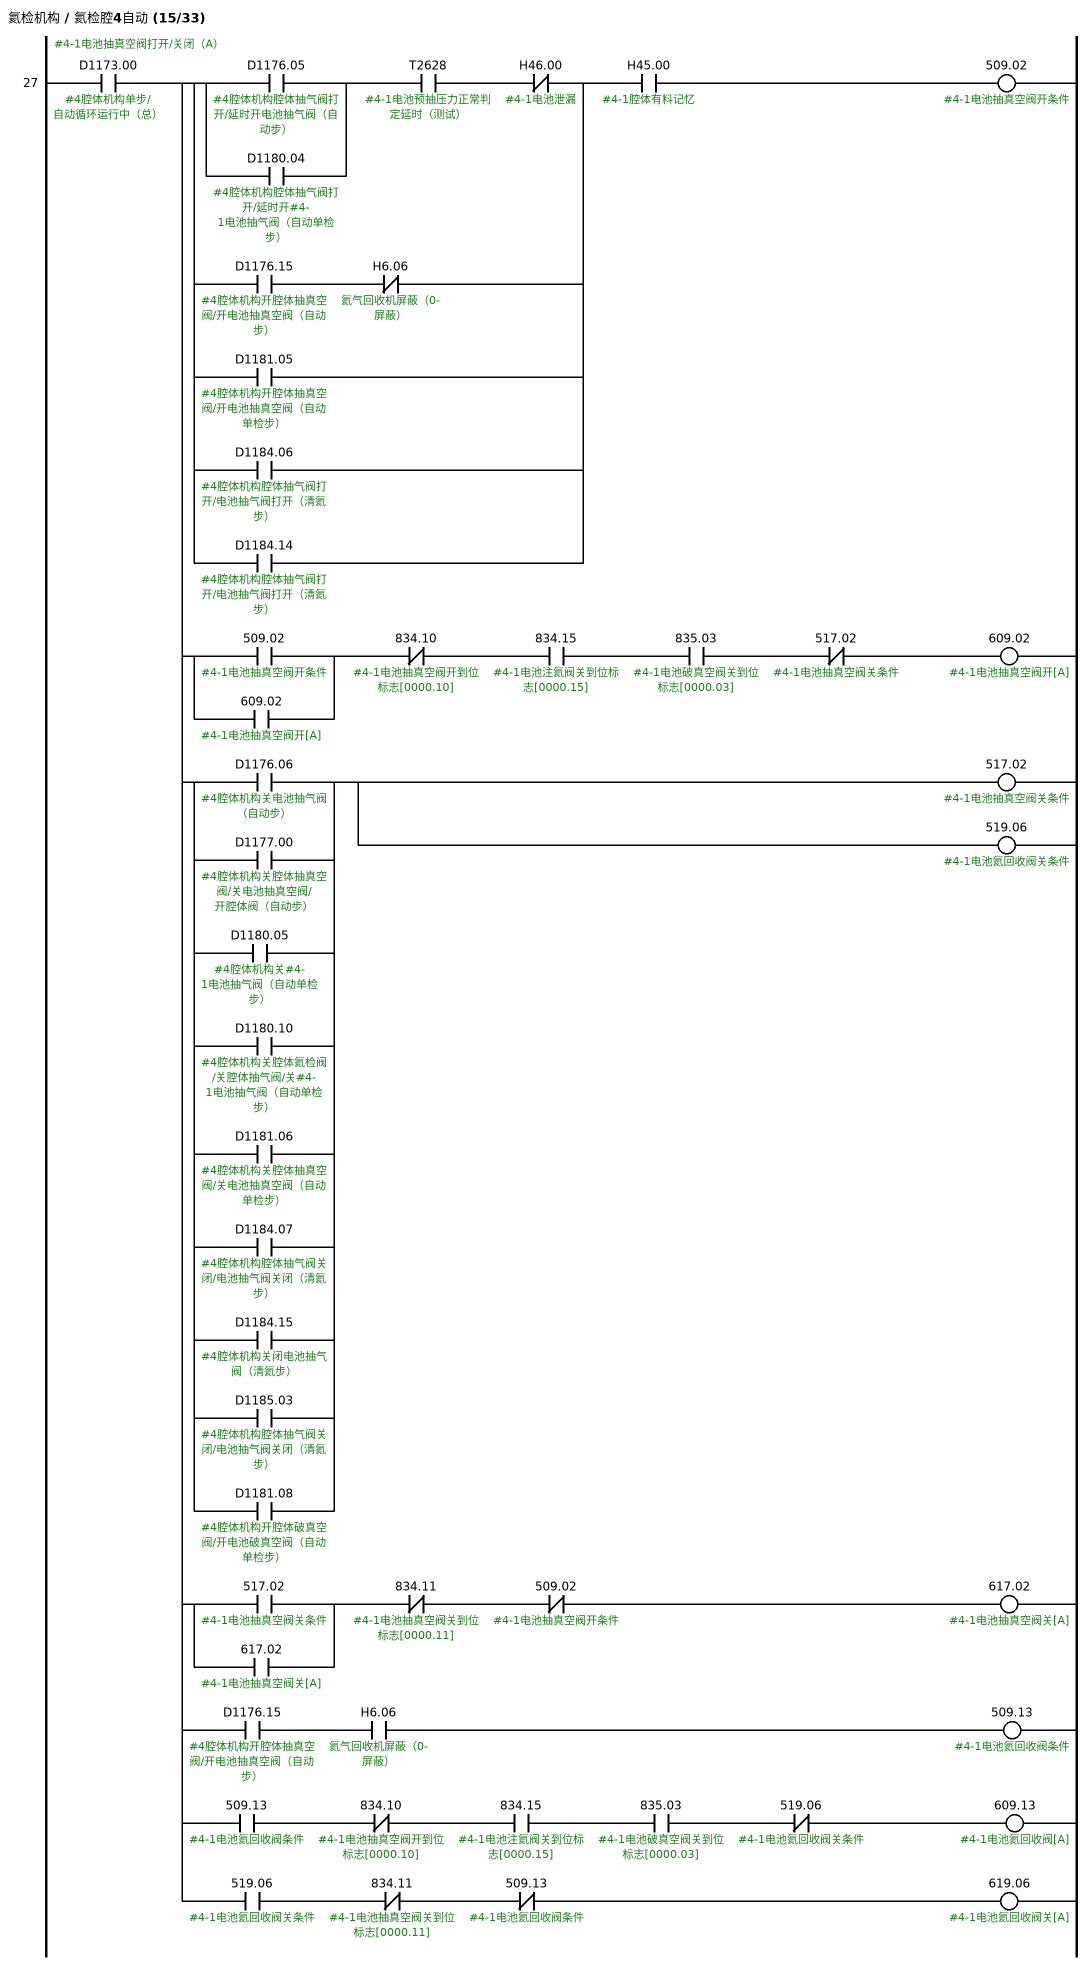
; rung 27: #4-1电池抽真空阀打开/关闭（A）
LD D1173.00  ; #4腔体机构单步/自动循环运行中（总）
OUT TR0
LD D1176.05  ; #4腔体机构腔体抽气阀打开/延时开电池抽气阀（自动步）
OR D1180.04  ; #4腔体机构腔体抽气阀打开/延时开#4-1电池抽气阀（自动单检步）
AND T2628  ; #4-1电池预抽压力正常判定延时（测试）
ANDNOT H46.00  ; #4-1电池泄漏
LD D1176.15  ; #4腔体机构开腔体抽真空阀/开电池抽真空阀（自动步）
ANDNOT H6.06  ; 氦气回收机屏蔽（0-屏蔽）
ORLD
OR D1181.05  ; #4腔体机构开腔体抽真空阀/开电池抽真空阀（自动单检步）
OR D1184.06  ; #4腔体机构腔体抽气阀打开/电池抽气阀打开（清氦步）
OR D1184.14  ; #4腔体机构腔体抽气阀打开/电池抽气阀打开（清氦步）
ANDLD
AND H45.00  ; #4-1腔体有料记忆
OUT 509.02  ; #4-1电池抽真空阀开条件
LD TR0
LD 509.02  ; #4-1电池抽真空阀开条件
OR 609.02  ; #4-1电池抽真空阀开[A]
ANDLD
ANDNOT 834.10  ; #4-1电池抽真空阀开到位标志[0000.10]
AND 834.15  ; #4-1电池注氦阀关到位标志[0000.15]
AND 835.03  ; #4-1电池破真空阀关到位标志[0000.03]
ANDNOT 517.02  ; #4-1电池抽真空阀关条件
OUT 609.02  ; #4-1电池抽真空阀开[A]
LD TR0
LD D1176.06  ; #4腔体机构关电池抽气阀（自动步）
OR D1177.00  ; #4腔体机构关腔体抽真空阀/关电池抽真空阀/开腔体阀（自动步）
OR D1180.05  ; #4腔体机构关#4-1电池抽气阀（自动单检步）
OR D1180.10  ; #4腔体机构关腔体氦检阀/关腔体抽气阀/关#4-1电池抽气阀（自动单检步）
OR D1181.06  ; #4腔体机构关腔体抽真空阀/关电池抽真空阀（自动单检步）
OR D1184.07  ; #4腔体机构腔体抽气阀关闭/电池抽气阀关闭（清氦步）
OR D1184.15  ; #4腔体机构关闭电池抽气阀（清氦步）
OR D1185.03  ; #4腔体机构腔体抽气阀关闭/电池抽气阀关闭（清氦步）
OR D1181.08  ; #4腔体机构开腔体破真空阀/开电池破真空阀（自动单检步）
ANDLD
OUT 517.02  ; #4-1电池抽真空阀关条件
OUT 519.06  ; #4-1电池氦回收阀关条件
LD TR0
LD 517.02  ; #4-1电池抽真空阀关条件
OR 617.02  ; #4-1电池抽真空阀关[A]
ANDLD
ANDNOT 834.11  ; #4-1电池抽真空阀关到位标志[0000.11]
ANDNOT 509.02  ; #4-1电池抽真空阀开条件
OUT 617.02  ; #4-1电池抽真空阀关[A]
LD TR0
AND D1176.15  ; #4腔体机构开腔体抽真空阀/开电池抽真空阀（自动步）
AND H6.06  ; 氦气回收机屏蔽（0-屏蔽）
OUT 509.13  ; #4-1电池氦回收阀条件
LD TR0
AND 509.13  ; #4-1电池氦回收阀条件
ANDNOT 834.10  ; #4-1电池抽真空阀开到位标志[0000.10]
AND 834.15  ; #4-1电池注氦阀关到位标志[0000.15]
AND 835.03  ; #4-1电池破真空阀关到位标志[0000.03]
ANDNOT 519.06  ; #4-1电池氦回收阀关条件
OUT 609.13  ; #4-1电池氦回收阀[A]
LD TR0
AND 519.06  ; #4-1电池氦回收阀关条件
ANDNOT 834.11  ; #4-1电池抽真空阀关到位标志[0000.11]
ANDNOT 509.13  ; #4-1电池氦回收阀条件
OUT 619.06  ; #4-1电池氦回收阀关[A]

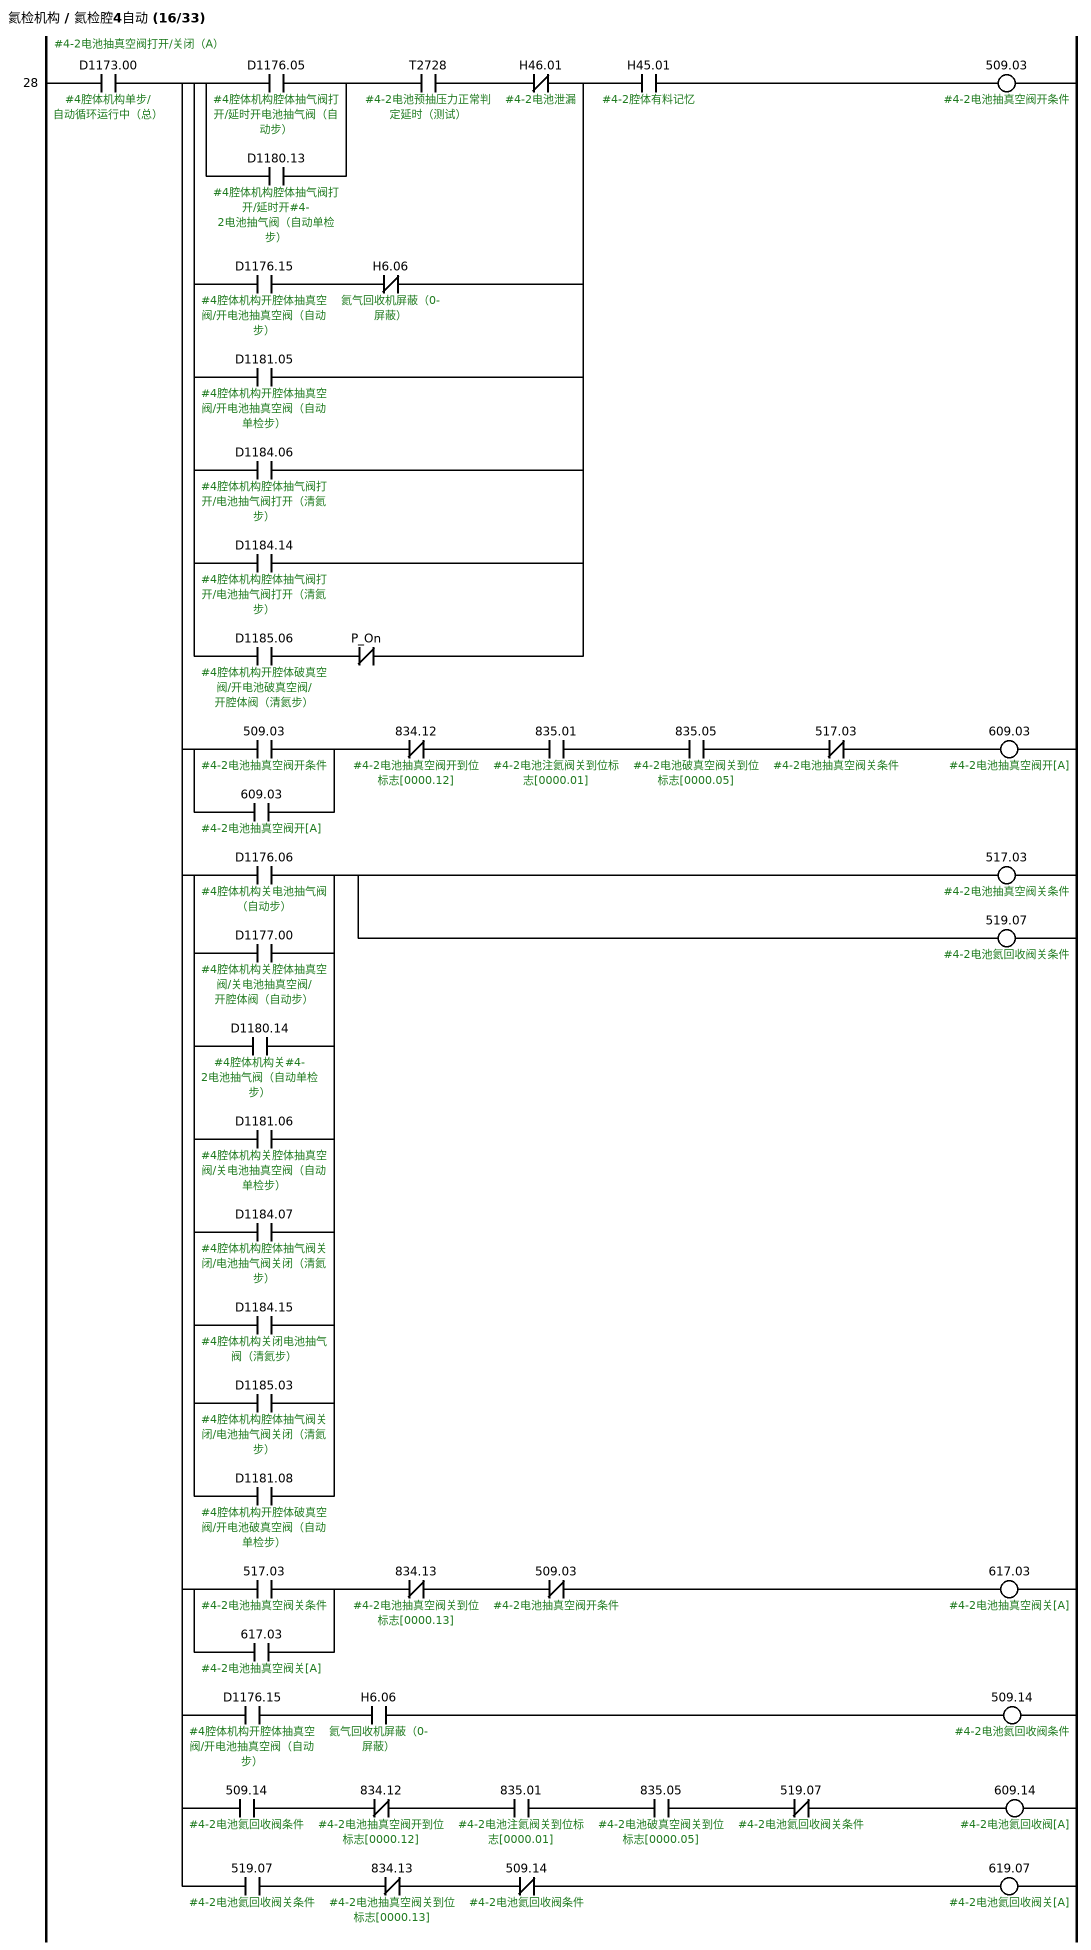
; rung 28: #4-2电池抽真空阀打开/关闭（A）
LD D1173.00  ; #4腔体机构单步/自动循环运行中（总）
OUT TR0
LD D1176.05  ; #4腔体机构腔体抽气阀打开/延时开电池抽气阀（自动步）
OR D1180.13  ; #4腔体机构腔体抽气阀打开/延时开#4-2电池抽气阀（自动单检步）
AND T2728  ; #4-2电池预抽压力正常判定延时（测试）
ANDNOT H46.01  ; #4-2电池泄漏
LD D1176.15  ; #4腔体机构开腔体抽真空阀/开电池抽真空阀（自动步）
ANDNOT H6.06  ; 氦气回收机屏蔽（0-屏蔽）
ORLD
OR D1181.05  ; #4腔体机构开腔体抽真空阀/开电池抽真空阀（自动单检步）
OR D1184.06  ; #4腔体机构腔体抽气阀打开/电池抽气阀打开（清氦步）
OR D1184.14  ; #4腔体机构腔体抽气阀打开/电池抽气阀打开（清氦步）
LD D1185.06  ; #4腔体机构开腔体破真空阀/开电池破真空阀/开腔体阀（清氦步）
ANDNOT P_On
ORLD
ANDLD
AND H45.01  ; #4-2腔体有料记忆
OUT 509.03  ; #4-2电池抽真空阀开条件
LD TR0
LD 509.03  ; #4-2电池抽真空阀开条件
OR 609.03  ; #4-2电池抽真空阀开[A]
ANDLD
ANDNOT 834.12  ; #4-2电池抽真空阀开到位标志[0000.12]
AND 835.01  ; #4-2电池注氦阀关到位标志[0000.01]
AND 835.05  ; #4-2电池破真空阀关到位标志[0000.05]
ANDNOT 517.03  ; #4-2电池抽真空阀关条件
OUT 609.03  ; #4-2电池抽真空阀开[A]
LD TR0
LD D1176.06  ; #4腔体机构关电池抽气阀（自动步）
OR D1177.00  ; #4腔体机构关腔体抽真空阀/关电池抽真空阀/开腔体阀（自动步）
OR D1180.14  ; #4腔体机构关#4-2电池抽气阀（自动单检步）
OR D1181.06  ; #4腔体机构关腔体抽真空阀/关电池抽真空阀（自动单检步）
OR D1184.07  ; #4腔体机构腔体抽气阀关闭/电池抽气阀关闭（清氦步）
OR D1184.15  ; #4腔体机构关闭电池抽气阀（清氦步）
OR D1185.03  ; #4腔体机构腔体抽气阀关闭/电池抽气阀关闭（清氦步）
OR D1181.08  ; #4腔体机构开腔体破真空阀/开电池破真空阀（自动单检步）
ANDLD
OUT 517.03  ; #4-2电池抽真空阀关条件
OUT 519.07  ; #4-2电池氦回收阀关条件
LD TR0
LD 517.03  ; #4-2电池抽真空阀关条件
OR 617.03  ; #4-2电池抽真空阀关[A]
ANDLD
ANDNOT 834.13  ; #4-2电池抽真空阀关到位标志[0000.13]
ANDNOT 509.03  ; #4-2电池抽真空阀开条件
OUT 617.03  ; #4-2电池抽真空阀关[A]
LD TR0
AND D1176.15  ; #4腔体机构开腔体抽真空阀/开电池抽真空阀（自动步）
AND H6.06  ; 氦气回收机屏蔽（0-屏蔽）
OUT 509.14  ; #4-2电池氦回收阀条件
LD TR0
AND 509.14  ; #4-2电池氦回收阀条件
ANDNOT 834.12  ; #4-2电池抽真空阀开到位标志[0000.12]
AND 835.01  ; #4-2电池注氦阀关到位标志[0000.01]
AND 835.05  ; #4-2电池破真空阀关到位标志[0000.05]
ANDNOT 519.07  ; #4-2电池氦回收阀关条件
OUT 609.14  ; #4-2电池氦回收阀[A]
LD TR0
AND 519.07  ; #4-2电池氦回收阀关条件
ANDNOT 834.13  ; #4-2电池抽真空阀关到位标志[0000.13]
ANDNOT 509.14  ; #4-2电池氦回收阀条件
OUT 619.07  ; #4-2电池氦回收阀关[A]

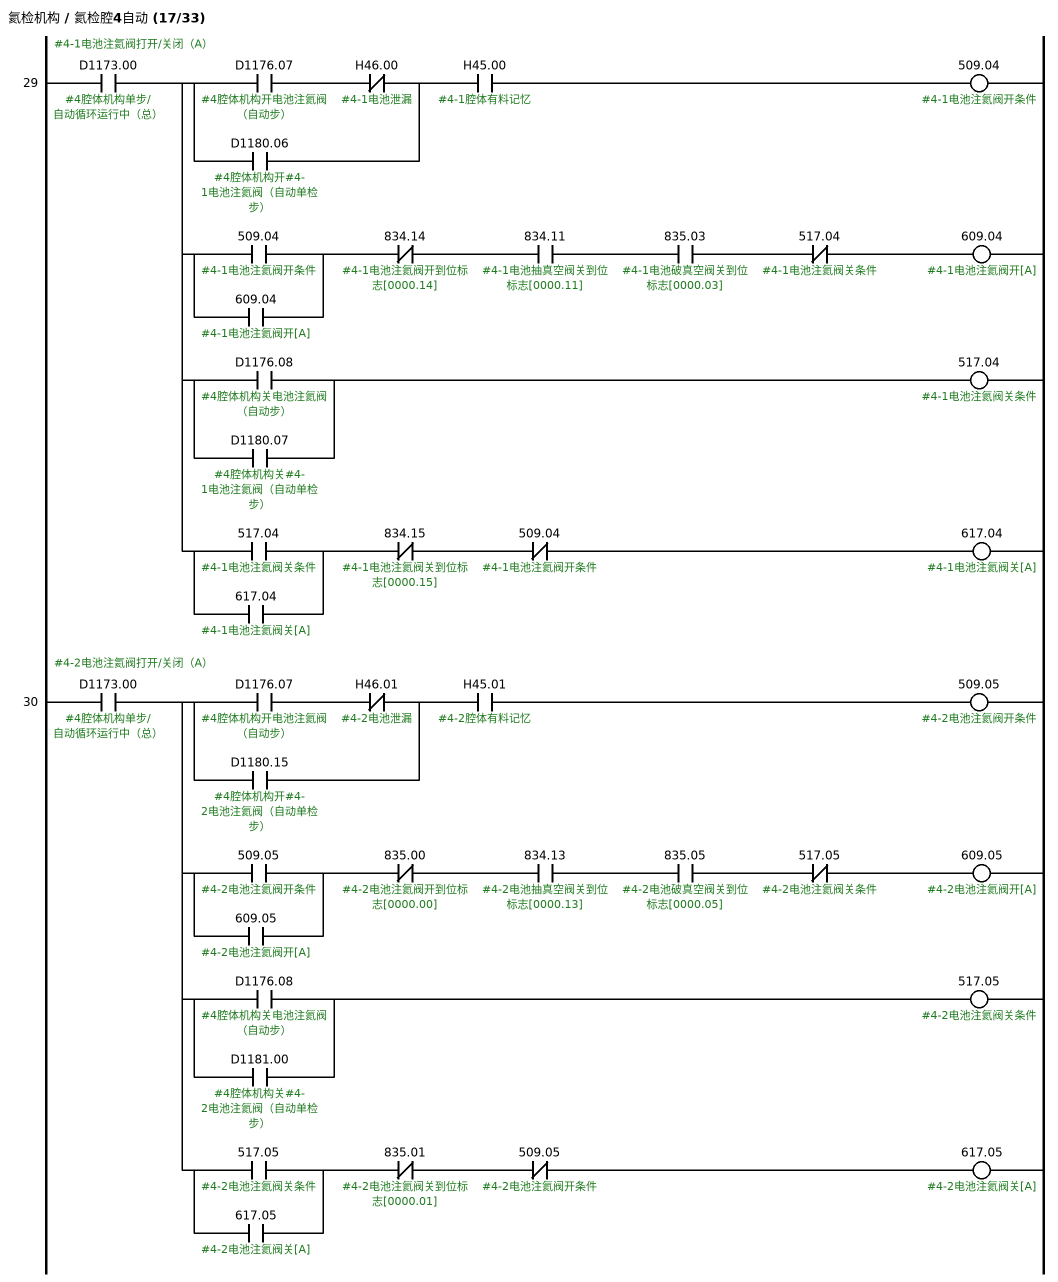
; rung 29: #4-1电池注氦阀打开/关闭（A）
LD D1173.00  ; #4腔体机构单步/自动循环运行中（总）
OUT TR0
LD D1176.07  ; #4腔体机构开电池注氦阀（自动步）
ANDNOT H46.00  ; #4-1电池泄漏
OR D1180.06  ; #4腔体机构开#4-1电池注氦阀（自动单检步）
ANDLD
AND H45.00  ; #4-1腔体有料记忆
OUT 509.04  ; #4-1电池注氦阀开条件
LD TR0
LD 509.04  ; #4-1电池注氦阀开条件
OR 609.04  ; #4-1电池注氦阀开[A]
ANDLD
ANDNOT 834.14  ; #4-1电池注氦阀开到位标志[0000.14]
AND 834.11  ; #4-1电池抽真空阀关到位标志[0000.11]
AND 835.03  ; #4-1电池破真空阀关到位标志[0000.03]
ANDNOT 517.04  ; #4-1电池注氦阀关条件
OUT 609.04  ; #4-1电池注氦阀开[A]
LD TR0
LD D1176.08  ; #4腔体机构关电池注氦阀（自动步）
OR D1180.07  ; #4腔体机构关#4-1电池注氦阀（自动单检步）
ANDLD
OUT 517.04  ; #4-1电池注氦阀关条件
LD TR0
LD 517.04  ; #4-1电池注氦阀关条件
OR 617.04  ; #4-1电池注氦阀关[A]
ANDLD
ANDNOT 834.15  ; #4-1电池注氦阀关到位标志[0000.15]
ANDNOT 509.04  ; #4-1电池注氦阀开条件
OUT 617.04  ; #4-1电池注氦阀关[A]
; rung 30: #4-2电池注氦阀打开/关闭（A）
LD D1173.00  ; #4腔体机构单步/自动循环运行中（总）
OUT TR0
LD D1176.07  ; #4腔体机构开电池注氦阀（自动步）
ANDNOT H46.01  ; #4-2电池泄漏
OR D1180.15  ; #4腔体机构开#4-2电池注氦阀（自动单检步）
ANDLD
AND H45.01  ; #4-2腔体有料记忆
OUT 509.05  ; #4-2电池注氦阀开条件
LD TR0
LD 509.05  ; #4-2电池注氦阀开条件
OR 609.05  ; #4-2电池注氦阀开[A]
ANDLD
ANDNOT 835.00  ; #4-2电池注氦阀开到位标志[0000.00]
AND 834.13  ; #4-2电池抽真空阀关到位标志[0000.13]
AND 835.05  ; #4-2电池破真空阀关到位标志[0000.05]
ANDNOT 517.05  ; #4-2电池注氦阀关条件
OUT 609.05  ; #4-2电池注氦阀开[A]
LD TR0
LD D1176.08  ; #4腔体机构关电池注氦阀（自动步）
OR D1181.00  ; #4腔体机构关#4-2电池注氦阀（自动单检步）
ANDLD
OUT 517.05  ; #4-2电池注氦阀关条件
LD TR0
LD 517.05  ; #4-2电池注氦阀关条件
OR 617.05  ; #4-2电池注氦阀关[A]
ANDLD
ANDNOT 835.01  ; #4-2电池注氦阀关到位标志[0000.01]
ANDNOT 509.05  ; #4-2电池注氦阀开条件
OUT 617.05  ; #4-2电池注氦阀关[A]

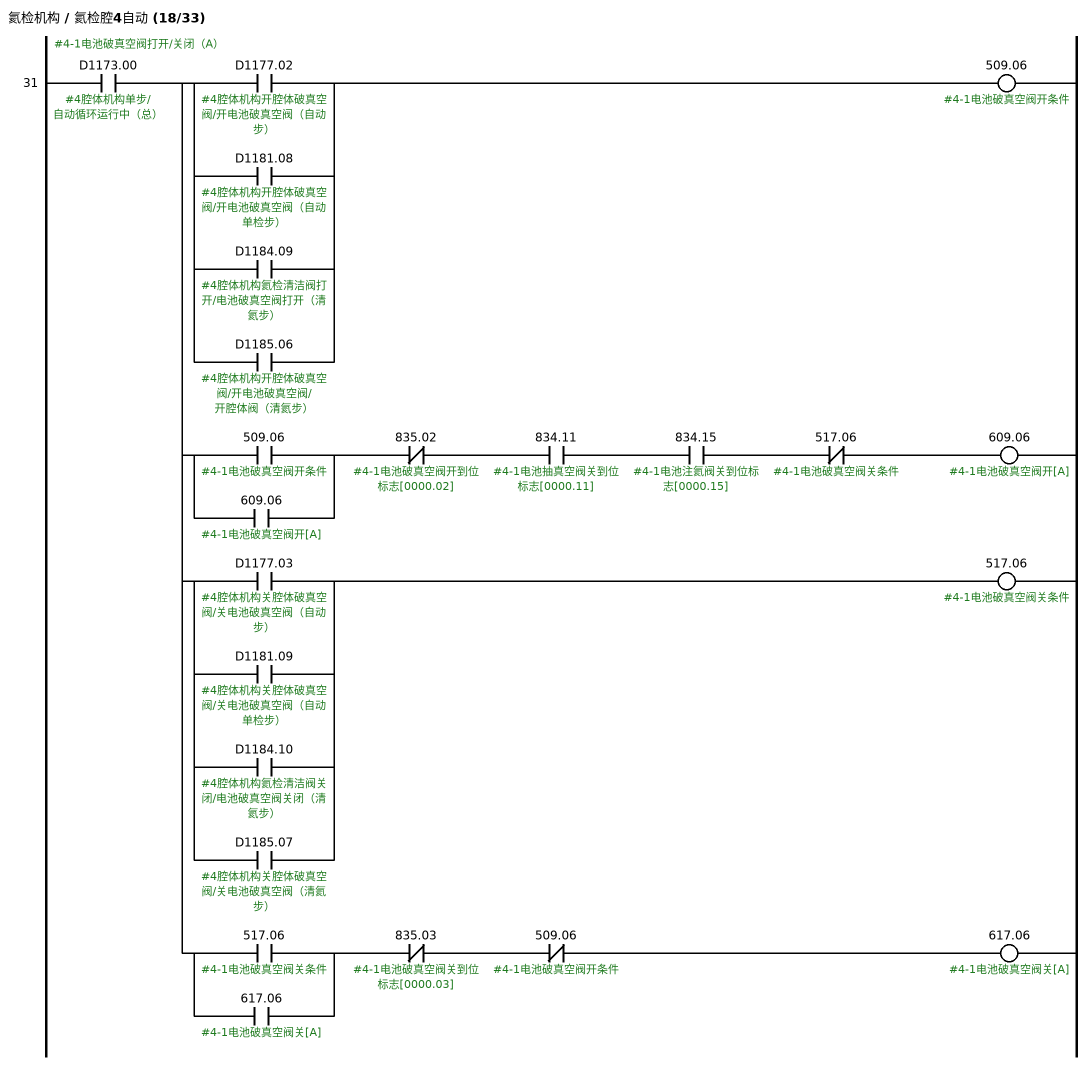
; rung 31: #4-1电池破真空阀打开/关闭（A）
LD D1173.00  ; #4腔体机构单步/自动循环运行中（总）
OUT TR0
LD D1177.02  ; #4腔体机构开腔体破真空阀/开电池破真空阀（自动步）
OR D1181.08  ; #4腔体机构开腔体破真空阀/开电池破真空阀（自动单检步）
OR D1184.09  ; #4腔体机构氦检清洁阀打开/电池破真空阀打开（清氦步）
OR D1185.06  ; #4腔体机构开腔体破真空阀/开电池破真空阀/开腔体阀（清氦步）
ANDLD
OUT 509.06  ; #4-1电池破真空阀开条件
LD TR0
LD 509.06  ; #4-1电池破真空阀开条件
OR 609.06  ; #4-1电池破真空阀开[A]
ANDLD
ANDNOT 835.02  ; #4-1电池破真空阀开到位标志[0000.02]
AND 834.11  ; #4-1电池抽真空阀关到位标志[0000.11]
AND 834.15  ; #4-1电池注氦阀关到位标志[0000.15]
ANDNOT 517.06  ; #4-1电池破真空阀关条件
OUT 609.06  ; #4-1电池破真空阀开[A]
LD TR0
LD D1177.03  ; #4腔体机构关腔体破真空阀/关电池破真空阀（自动步）
OR D1181.09  ; #4腔体机构关腔体破真空阀/关电池破真空阀（自动单检步）
OR D1184.10  ; #4腔体机构氦检清洁阀关闭/电池破真空阀关闭（清氦步）
OR D1185.07  ; #4腔体机构关腔体破真空阀/关电池破真空阀（清氦步）
ANDLD
OUT 517.06  ; #4-1电池破真空阀关条件
LD TR0
LD 517.06  ; #4-1电池破真空阀关条件
OR 617.06  ; #4-1电池破真空阀关[A]
ANDLD
ANDNOT 835.03  ; #4-1电池破真空阀关到位标志[0000.03]
ANDNOT 509.06  ; #4-1电池破真空阀开条件
OUT 617.06  ; #4-1电池破真空阀关[A]

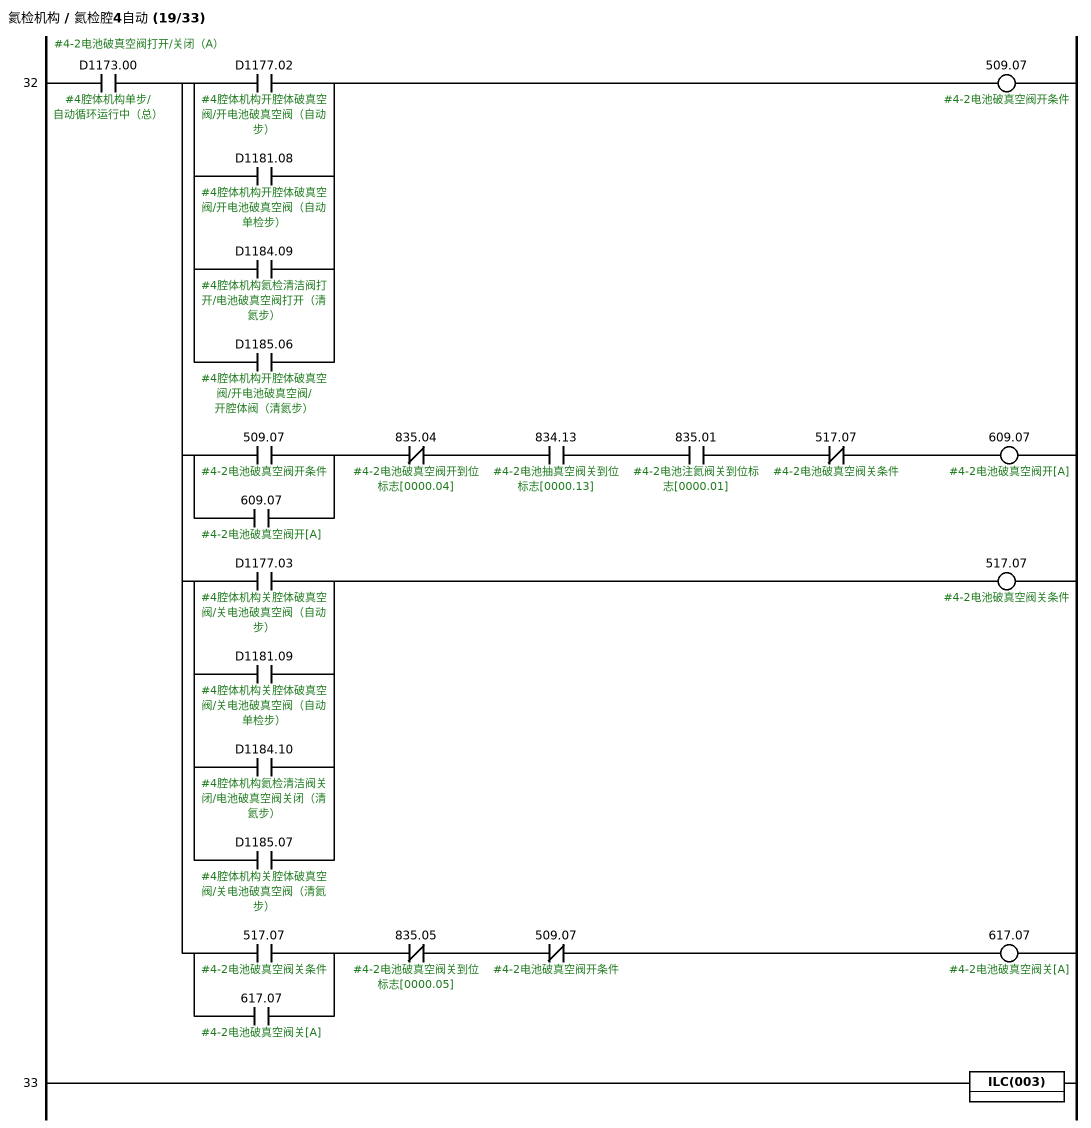
; rung 32: #4-2电池破真空阀打开/关闭（A）
LD D1173.00  ; #4腔体机构单步/自动循环运行中（总）
OUT TR0
LD D1177.02  ; #4腔体机构开腔体破真空阀/开电池破真空阀（自动步）
OR D1181.08  ; #4腔体机构开腔体破真空阀/开电池破真空阀（自动单检步）
OR D1184.09  ; #4腔体机构氦检清洁阀打开/电池破真空阀打开（清氦步）
OR D1185.06  ; #4腔体机构开腔体破真空阀/开电池破真空阀/开腔体阀（清氦步）
ANDLD
OUT 509.07  ; #4-2电池破真空阀开条件
LD TR0
LD 509.07  ; #4-2电池破真空阀开条件
OR 609.07  ; #4-2电池破真空阀开[A]
ANDLD
ANDNOT 835.04  ; #4-2电池破真空阀开到位标志[0000.04]
AND 834.13  ; #4-2电池抽真空阀关到位标志[0000.13]
AND 835.01  ; #4-2电池注氦阀关到位标志[0000.01]
ANDNOT 517.07  ; #4-2电池破真空阀关条件
OUT 609.07  ; #4-2电池破真空阀开[A]
LD TR0
LD D1177.03  ; #4腔体机构关腔体破真空阀/关电池破真空阀（自动步）
OR D1181.09  ; #4腔体机构关腔体破真空阀/关电池破真空阀（自动单检步）
OR D1184.10  ; #4腔体机构氦检清洁阀关闭/电池破真空阀关闭（清氦步）
OR D1185.07  ; #4腔体机构关腔体破真空阀/关电池破真空阀（清氦步）
ANDLD
OUT 517.07  ; #4-2电池破真空阀关条件
LD TR0
LD 517.07  ; #4-2电池破真空阀关条件
OR 617.07  ; #4-2电池破真空阀关[A]
ANDLD
ANDNOT 835.05  ; #4-2电池破真空阀关到位标志[0000.05]
ANDNOT 509.07  ; #4-2电池破真空阀开条件
OUT 617.07  ; #4-2电池破真空阀关[A]
; rung 33
ILC(003)

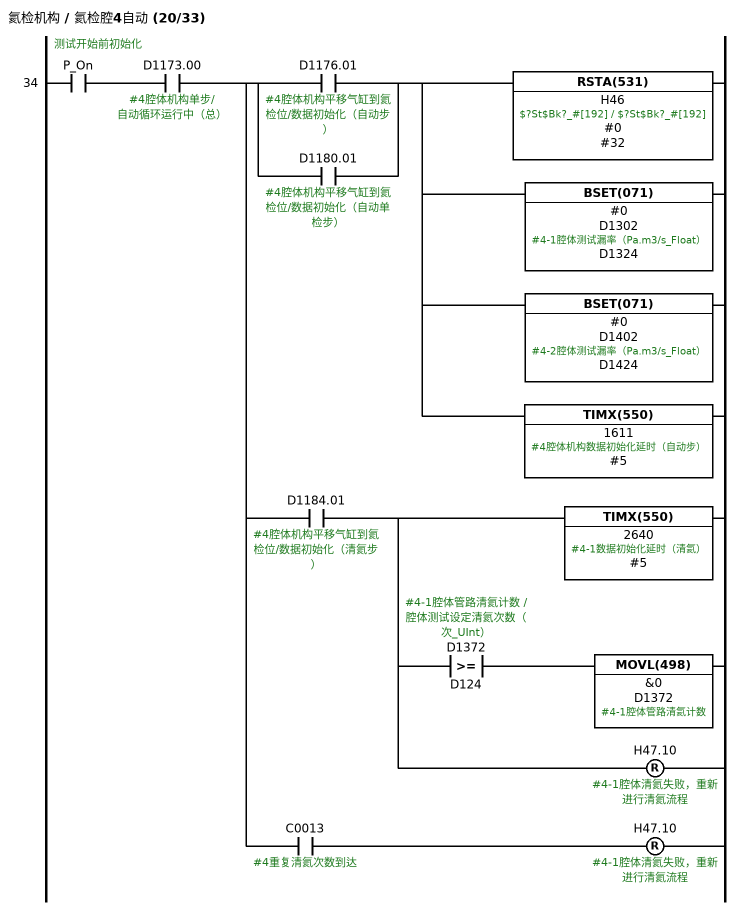
; rung 34: 测试开始前初始化
LD P_On
AND D1173.00  ; #4腔体机构单步/自动循环运行中（总）
OUT TR0
LD D1176.01  ; #4腔体机构平移气缸到氦检位/数据初始化（自动步）
OR D1180.01  ; #4腔体机构平移气缸到氦检位/数据初始化（自动单检步）
ANDLD
RSTA(531) H46 #0 #32  ; $?St$Bk?_#[192] / $?St$Bk?_#[192]
BSET(071) #0 D1302 D1324  ; #4-1腔体测试漏率（Pa.m3/s_Float）
BSET(071) #0 D1402 D1424  ; #4-2腔体测试漏率（Pa.m3/s_Float）
TIMX(550) 1611 #5  ; #4腔体机构数据初始化延时（自动步）
LD TR0
AND D1184.01  ; #4腔体机构平移气缸到氦检位/数据初始化（清氦步）
OUT TR1
TIMX(550) 2640 #5  ; #4-1数据初始化延时（清氦）
AND>=(325) D1372 D124  ; #4-1腔体管路清氦计数, 腔体测试设定清氦次数（次_UInt）
MOVL(498) &0 D1372  ; #4-1腔体管路清氦计数
LD TR1
RSET H47.10  ; #4-1腔体清氦失败，重新进行清氦流程
LD TR0
AND C0013  ; #4重复清氦次数到达
RSET H47.10  ; #4-1腔体清氦失败，重新进行清氦流程

